   1:  PR[GP1:91,1] = PR[GP1:90,1] + -15.770;
   1:  PR[GP1:91,2] = PR[GP1:90,2] + -15.065;
   1:L PR[91] 10mm/sec CNT100;
   1:  PR[GP1:91,1] = PR[GP1:90,1] + -15.094;
   1:  PR[GP1:91,2] = PR[GP1:90,2] + -15.115;
   1:  PR[GP1:91,3] = PR[GP1:90,3] + 48.400;
   1:L PR[91] 10mm/sec CNT100;
   1:  PR[GP1:91,1] = PR[GP1:90,1] + -12.204;
   1:  PR[GP1:91,2] = PR[GP1:90,2] + -18.068;
   1:L PR[91] 10mm/sec CNT100;
   1:  PR[GP1:91,1] = PR[GP1:90,1] + -12.047;
   1:  PR[GP1:91,2] = PR[GP1:90,2] + -18.203;
   1:L PR[91] 10mm/sec CNT100;
   1:  PR[GP1:91,1] = PR[GP1:90,1] + -10.939;
   1:  PR[GP1:91,2] = PR[GP1:90,2] + -18.959;
   1:L PR[91] 10mm/sec CNT100;
   1:  PR[GP1:91,1] = PR[GP1:90,1] + -8.236;
   1:  PR[GP1:91,2] = PR[GP1:90,2] + -20.991;
   1:L PR[91] 10mm/sec CNT100;
   1:  PR[GP1:91,1] = PR[GP1:90,1] + -7.444;
   1:  PR[GP1:91,2] = PR[GP1:90,2] + -21.525;
   1:L PR[91] 10mm/sec CNT100;
   1:  PR[GP1:91,1] = PR[GP1:90,1] + -4.180;
   1:  PR[GP1:91,2] = PR[GP1:90,2] + -23.163;
   1:L PR[91] 10mm/sec CNT100;
   1:  PR[GP1:91,1] = PR[GP1:90,1] + -1.871;
   1:  PR[GP1:91,2] = PR[GP1:90,2] + -24.171;
   1:L PR[91] 10mm/sec CNT100;
   1:  PR[GP1:91,1] = PR[GP1:90,1] + 0.209;
   1:  PR[GP1:91,2] = PR[GP1:90,2] + -24.790;
   1:L PR[91] 10mm/sec CNT100;
   1:  PR[GP1:91,1] = PR[GP1:90,1] + 4.204;
   1:  PR[GP1:91,2] = PR[GP1:90,2] + -25.728;
   1:L PR[91] 10mm/sec CNT100;
   1:  PR[GP1:91,1] = PR[GP1:90,1] + 4.832;
   1:  PR[GP1:91,2] = PR[GP1:90,2] + -25.796;
   1:L PR[91] 10mm/sec CNT100;
   1:  PR[GP1:91,1] = PR[GP1:90,1] + 7.181;
   1:  PR[GP1:91,2] = PR[GP1:90,2] + -25.893;
   1:L PR[91] 10mm/sec CNT100;
   1:  PR[GP1:91,1] = PR[GP1:90,1] + 9.648;
   1:  PR[GP1:91,2] = PR[GP1:90,2] + -26.131;
   1:L PR[91] 10mm/sec CNT100;
   1:  PR[GP1:91,1] = PR[GP1:90,1] + 9.702;
   1:  PR[GP1:91,2] = PR[GP1:90,2] + -26.096;
   1:L PR[91] 10mm/sec CNT100;
   1:  PR[GP1:91,1] = PR[GP1:90,1] + 10.831;
   1:  PR[GP1:91,2] = PR[GP1:90,2] + -26.181;
   1:L PR[91] 10mm/sec CNT100;
   1:  PR[GP1:91,1] = PR[GP1:90,1] + 13.329;
   1:  PR[GP1:91,2] = PR[GP1:90,2] + -26.259;
   1:L PR[91] 10mm/sec CNT100;
   1:  PR[GP1:91,1] = PR[GP1:90,1] + 13.483;
   1:  PR[GP1:91,2] = PR[GP1:90,2] + -26.256;
   1:L PR[91] 10mm/sec CNT100;
   1:  PR[GP1:91,1] = PR[GP1:90,1] + 15.783;
   1:  PR[GP1:91,2] = PR[GP1:90,2] + -26.009;
   1:L PR[91] 10mm/sec CNT100;
   1:  PR[GP1:91,1] = PR[GP1:90,1] + 16.739;
   1:  PR[GP1:91,2] = PR[GP1:90,2] + -25.829;
   1:L PR[91] 10mm/sec CNT100;
   1:  PR[GP1:91,1] = PR[GP1:90,1] + 18.227;
   1:  PR[GP1:91,2] = PR[GP1:90,2] + -25.423;
   1:L PR[91] 10mm/sec CNT100;
   1:  PR[GP1:91,1] = PR[GP1:90,1] + 19.830;
   1:  PR[GP1:91,2] = PR[GP1:90,2] + -24.829;
   1:L PR[91] 10mm/sec CNT100;
   1:  PR[GP1:91,1] = PR[GP1:90,1] + 20.623;
   1:  PR[GP1:91,2] = PR[GP1:90,2] + -24.464;
   1:L PR[91] 10mm/sec CNT100;
   1:  PR[GP1:91,1] = PR[GP1:90,1] + 22.593;
   1:  PR[GP1:91,2] = PR[GP1:90,2] + -23.304;
   1:L PR[91] 10mm/sec CNT100;
   1:  PR[GP1:91,1] = PR[GP1:90,1] + 22.905;
   1:  PR[GP1:91,2] = PR[GP1:90,2] + -23.089;
   1:L PR[91] 10mm/sec CNT100;
   1:  PR[GP1:91,1] = PR[GP1:90,1] + 24.893;
   1:  PR[GP1:91,2] = PR[GP1:90,2] + -21.368;
   1:L PR[91] 10mm/sec CNT100;
   1:  PR[GP1:91,1] = PR[GP1:90,1] + 24.984;
   1:  PR[GP1:91,2] = PR[GP1:90,2] + -21.279;
   1:L PR[91] 10mm/sec CNT100;
   1:  PR[GP1:91,1] = PR[GP1:90,1] + 26.658;
   1:  PR[GP1:91,2] = PR[GP1:90,2] + -19.173;
   1:L PR[91] 10mm/sec CNT100;
   1:  PR[GP1:91,1] = PR[GP1:90,1] + 26.752;
   1:  PR[GP1:91,2] = PR[GP1:90,2] + -19.040;
   1:L PR[91] 10mm/sec CNT100;
   1:  PR[GP1:91,1] = PR[GP1:90,1] + 27.909;
   1:  PR[GP1:91,2] = PR[GP1:90,2] + -16.870;
   1:L PR[91] 10mm/sec CNT100;
   1:  PR[GP1:91,1] = PR[GP1:90,1] + 28.113;
   1:  PR[GP1:91,2] = PR[GP1:90,2] + -16.441;
   1:L PR[91] 10mm/sec CNT100;
   1:  PR[GP1:91,1] = PR[GP1:90,1] + 28.728;
   1:  PR[GP1:91,2] = PR[GP1:90,2] + -14.577;
   1:L PR[91] 10mm/sec CNT100;
   1:  PR[GP1:91,1] = PR[GP1:90,1] + 29.009;
   1:  PR[GP1:91,2] = PR[GP1:90,2] + -13.612;
   1:L PR[91] 10mm/sec CNT100;
   1:  PR[GP1:91,1] = PR[GP1:90,1] + 29.195;
   1:  PR[GP1:91,2] = PR[GP1:90,2] + -12.364;
   1:L PR[91] 10mm/sec CNT100;
   1:  PR[GP1:91,1] = PR[GP1:90,1] + 29.399;
   1:  PR[GP1:91,2] = PR[GP1:90,2] + -10.701;
   1:L PR[91] 10mm/sec CNT100;
   1:  PR[GP1:91,1] = PR[GP1:90,1] + 29.327;
   1:  PR[GP1:91,2] = PR[GP1:90,2] + -9.105;
   1:L PR[91] 10mm/sec CNT100;
   1:  PR[GP1:91,1] = PR[GP1:90,1] + 29.296;
   1:  PR[GP1:91,2] = PR[GP1:90,2] + -7.776;
   1:L PR[91] 10mm/sec CNT100;
   1:  PR[GP1:91,1] = PR[GP1:90,1] + 28.542;
   1:  PR[GP1:91,2] = PR[GP1:90,2] + -3.810;
   1:L PR[91] 10mm/sec CNT100;
   1:  PR[GP1:91,1] = PR[GP1:90,1] + 27.855;
   1:  PR[GP1:91,2] = PR[GP1:90,2] + -2.041;
   1:L PR[91] 10mm/sec CNT100;
   1:  PR[GP1:91,1] = PR[GP1:90,1] + 27.141;
   1:  PR[GP1:91,2] = PR[GP1:90,2] + -0.046;
   1:L PR[91] 10mm/sec CNT100;
   1:  PR[GP1:91,1] = PR[GP1:90,1] + 26.192;
   1:  PR[GP1:91,2] = PR[GP1:90,2] + 1.584;
   1:L PR[91] 10mm/sec CNT100;
   1:  PR[GP1:91,1] = PR[GP1:90,1] + 25.121;
   1:  PR[GP1:91,2] = PR[GP1:90,2] + 3.337;
   1:L PR[91] 10mm/sec CNT100;
   1:  PR[GP1:91,1] = PR[GP1:90,1] + 22.561;
   1:  PR[GP1:91,2] = PR[GP1:90,2] + 6.231;
   1:L PR[91] 10mm/sec CNT100;
   1:  PR[GP1:91,1] = PR[GP1:90,1] + 19.685;
   1:  PR[GP1:91,2] = PR[GP1:90,2] + 8.504;
   1:L PR[91] 10mm/sec CNT100;
   1:  PR[GP1:91,1] = PR[GP1:90,1] + 17.372;
   1:  PR[GP1:91,2] = PR[GP1:90,2] + 9.702;
   1:L PR[91] 10mm/sec CNT100;
   1:  PR[GP1:91,1] = PR[GP1:90,1] + 16.514;
   1:  PR[GP1:91,2] = PR[GP1:90,2] + 10.131;
   1:L PR[91] 10mm/sec CNT100;
   1:  PR[GP1:91,1] = PR[GP1:90,1] + 13.120;
   1:  PR[GP1:91,2] = PR[GP1:90,2] + 11.100;
   1:L PR[91] 10mm/sec CNT100;
   1:  PR[GP1:91,1] = PR[GP1:90,1] + 9.749;
   1:  PR[GP1:91,2] = PR[GP1:90,2] + 11.359;
   1:L PR[91] 10mm/sec CNT100;
   1:  PR[GP1:91,1] = PR[GP1:90,1] + 7.022;
   1:  PR[GP1:91,2] = PR[GP1:90,2] + 11.063;
   1:L PR[91] 10mm/sec CNT100;
   1:  PR[GP1:91,1] = PR[GP1:90,1] + 6.312;
   1:  PR[GP1:91,2] = PR[GP1:90,2] + 10.967;
   1:L PR[91] 10mm/sec CNT100;
   1:  PR[GP1:91,1] = PR[GP1:90,1] + 5.302;
   1:  PR[GP1:91,2] = PR[GP1:90,2] + 10.725;
   1:L PR[91] 10mm/sec CNT100;
   1:  PR[GP1:91,1] = PR[GP1:90,1] + 4.246;
   1:  PR[GP1:91,2] = PR[GP1:90,2] + 10.670;
   1:L PR[91] 10mm/sec CNT100;
   1:  PR[GP1:91,1] = PR[GP1:90,1] + 3.038;
   1:  PR[GP1:91,2] = PR[GP1:90,2] + 10.819;
   1:L PR[91] 10mm/sec CNT100;
   1:  PR[GP1:91,1] = PR[GP1:90,1] + 2.391;
   1:  PR[GP1:91,2] = PR[GP1:90,2] + 10.872;
   1:L PR[91] 10mm/sec CNT100;
   1:  PR[GP1:91,1] = PR[GP1:90,1] + 0.714;
   1:  PR[GP1:91,2] = PR[GP1:90,2] + 10.880;
   1:L PR[91] 10mm/sec CNT100;
   1:  PR[GP1:91,1] = PR[GP1:90,1] + -2.362;
   1:  PR[GP1:91,2] = PR[GP1:90,2] + 10.966;
   1:L PR[91] 10mm/sec CNT100;
   1:  PR[GP1:91,1] = PR[GP1:90,1] + -2.905;
   1:  PR[GP1:91,2] = PR[GP1:90,2] + 10.871;
   1:L PR[91] 10mm/sec CNT100;
   1:  PR[GP1:91,1] = PR[GP1:90,1] + -5.532;
   1:  PR[GP1:91,2] = PR[GP1:90,2] + 10.488;
   1:L PR[91] 10mm/sec CNT100;
   1:  PR[GP1:91,1] = PR[GP1:90,1] + -6.743;
   1:  PR[GP1:91,2] = PR[GP1:90,2] + 10.278;
   1:L PR[91] 10mm/sec CNT100;
   1:  PR[GP1:91,1] = PR[GP1:90,1] + -10.509;
   1:  PR[GP1:91,2] = PR[GP1:90,2] + 8.898;
   1:L PR[91] 10mm/sec CNT100;
   1:  PR[GP1:91,1] = PR[GP1:90,1] + -11.154;
   1:  PR[GP1:91,2] = PR[GP1:90,2] + 8.565;
   1:L PR[91] 10mm/sec CNT100;
   1:  PR[GP1:91,1] = PR[GP1:90,1] + -13.410;
   1:  PR[GP1:91,2] = PR[GP1:90,2] + 7.155;
   1:L PR[91] 10mm/sec CNT100;
   1:  PR[GP1:91,1] = PR[GP1:90,1] + -14.230;
   1:  PR[GP1:91,2] = PR[GP1:90,2] + 6.566;
   1:L PR[91] 10mm/sec CNT100;
   1:  PR[GP1:91,1] = PR[GP1:90,1] + -15.076;
   1:  PR[GP1:91,2] = PR[GP1:90,2] + 5.725;
   1:L PR[91] 10mm/sec CNT100;
   1:  PR[GP1:91,1] = PR[GP1:90,1] + -16.449;
   1:  PR[GP1:91,2] = PR[GP1:90,2] + 4.321;
   1:L PR[91] 10mm/sec CNT100;
   1:  PR[GP1:91,1] = PR[GP1:90,1] + -17.220;
   1:  PR[GP1:91,2] = PR[GP1:90,2] + 3.226;
   1:L PR[91] 10mm/sec CNT100;
   1:  PR[GP1:91,1] = PR[GP1:90,1] + -18.002;
   1:  PR[GP1:91,2] = PR[GP1:90,2] + 1.859;
   1:L PR[91] 10mm/sec CNT100;
   1:  PR[GP1:91,1] = PR[GP1:90,1] + -18.613;
   1:  PR[GP1:91,2] = PR[GP1:90,2] + 0.586;
   1:L PR[91] 10mm/sec CNT100;
   1:  PR[GP1:91,1] = PR[GP1:90,1] + -18.999;
   1:  PR[GP1:91,2] = PR[GP1:90,2] + -0.732;
   1:L PR[91] 10mm/sec CNT100;
   1:  PR[GP1:91,1] = PR[GP1:90,1] + -19.382;
   1:  PR[GP1:91,2] = PR[GP1:90,2] + -2.113;
   1:L PR[91] 10mm/sec CNT100;
   1:  PR[GP1:91,1] = PR[GP1:90,1] + -19.503;
   1:  PR[GP1:91,2] = PR[GP1:90,2] + -3.246;
   1:L PR[91] 10mm/sec CNT100;
   1:  PR[GP1:91,1] = PR[GP1:90,1] + -19.408;
   1:  PR[GP1:91,2] = PR[GP1:90,2] + -4.297;
   1:L PR[91] 10mm/sec CNT100;
   1:  PR[GP1:91,1] = PR[GP1:90,1] + -19.357;
   1:  PR[GP1:91,2] = PR[GP1:90,2] + -5.931;
   1:L PR[91] 10mm/sec CNT100;
   1:  PR[GP1:91,1] = PR[GP1:90,1] + -18.969;
   1:  PR[GP1:91,2] = PR[GP1:90,2] + -7.508;
   1:L PR[91] 10mm/sec CNT100;
   1:  PR[GP1:91,1] = PR[GP1:90,1] + -18.897;
   1:  PR[GP1:91,2] = PR[GP1:90,2] + -7.858;
   1:L PR[91] 10mm/sec CNT100;
   1:  PR[GP1:91,1] = PR[GP1:90,1] + -18.309;
   1:  PR[GP1:91,2] = PR[GP1:90,2] + -9.744;
   1:L PR[91] 10mm/sec CNT100;
   1:  PR[GP1:91,1] = PR[GP1:90,1] + -17.743;
   1:  PR[GP1:91,2] = PR[GP1:90,2] + -11.092;
   1:L PR[91] 10mm/sec CNT100;
   1:  PR[GP1:91,1] = PR[GP1:90,1] + -16.255;
   1:  PR[GP1:91,2] = PR[GP1:90,2] + -13.561;
   1:L PR[91] 10mm/sec CNT100;
   1:  PR[GP1:91,1] = PR[GP1:90,1] + -15.677;
   1:  PR[GP1:91,2] = PR[GP1:90,2] + -14.456;
   1:L PR[91] 10mm/sec CNT100;
   1:  PR[GP1:91,1] = PR[GP1:90,1] + -14.775;
   1:  PR[GP1:91,2] = PR[GP1:90,2] + -14.761;
   1:  PR[GP1:91,3] = PR[GP1:90,3] + 49.500;
   1:L PR[91] 10mm/sec CNT100;
   1:  PR[GP1:91,1] = PR[GP1:90,1] + -14.417;
   1:  PR[GP1:91,2] = PR[GP1:90,2] + -15.165;
   1:L PR[91] 10mm/sec CNT100;
   1:  PR[GP1:91,1] = PR[GP1:90,1] + -11.762;
   1:  PR[GP1:91,2] = PR[GP1:90,2] + -17.878;
   1:L PR[91] 10mm/sec CNT100;
   1:  PR[GP1:91,1] = PR[GP1:90,1] + -11.164;
   1:  PR[GP1:91,2] = PR[GP1:90,2] + -18.525;
   1:L PR[91] 10mm/sec CNT100;
   1:  PR[GP1:91,1] = PR[GP1:90,1] + -7.674;
   1:  PR[GP1:91,2] = PR[GP1:90,2] + -21.149;
   1:L PR[91] 10mm/sec CNT100;
   1:  PR[GP1:91,1] = PR[GP1:90,1] + -6.405;
   1:  PR[GP1:91,2] = PR[GP1:90,2] + -22.005;
   1:L PR[91] 10mm/sec CNT100;
   1:  PR[GP1:91,1] = PR[GP1:90,1] + -3.644;
   1:  PR[GP1:91,2] = PR[GP1:90,2] + -23.391;
   1:L PR[91] 10mm/sec CNT100;
   1:  PR[GP1:91,1] = PR[GP1:90,1] + -0.787;
   1:  PR[GP1:91,2] = PR[GP1:90,2] + -24.637;
   1:L PR[91] 10mm/sec CNT100;
   1:  PR[GP1:91,1] = PR[GP1:90,1] + 0.739;
   1:  PR[GP1:91,2] = PR[GP1:90,2] + -25.091;
   1:L PR[91] 10mm/sec CNT100;
   1:  PR[GP1:91,1] = PR[GP1:90,1] + 5.307;
   1:  PR[GP1:91,2] = PR[GP1:90,2] + -26.164;
   1:L PR[91] 10mm/sec CNT100;
   1:  PR[GP1:91,1] = PR[GP1:90,1] + 5.772;
   1:  PR[GP1:91,2] = PR[GP1:90,2] + -26.190;
   1:L PR[91] 10mm/sec CNT100;
   1:  PR[GP1:91,1] = PR[GP1:90,1] + 10.401;
   1:  PR[GP1:91,2] = PR[GP1:90,2] + -26.636;
   1:L PR[91] 10mm/sec CNT100;
   1:  PR[GP1:91,1] = PR[GP1:90,1] + 10.434;
   1:  PR[GP1:91,2] = PR[GP1:90,2] + -26.619;
   1:L PR[91] 10mm/sec CNT100;
   1:  PR[GP1:91,1] = PR[GP1:90,1] + 10.667;
   1:  PR[GP1:91,2] = PR[GP1:90,2] + -26.588;
   1:L PR[91] 10mm/sec CNT100;
   1:  PR[GP1:91,1] = PR[GP1:90,1] + 13.212;
   1:  PR[GP1:91,2] = PR[GP1:90,2] + -26.704;
   1:L PR[91] 10mm/sec CNT100;
   1:  PR[GP1:91,1] = PR[GP1:90,1] + 14.461;
   1:  PR[GP1:91,2] = PR[GP1:90,2] + -26.677;
   1:L PR[91] 10mm/sec CNT100;
   1:  PR[GP1:91,1] = PR[GP1:90,1] + 15.692;
   1:  PR[GP1:91,2] = PR[GP1:90,2] + -26.545;
   1:L PR[91] 10mm/sec CNT100;
   1:  PR[GP1:91,1] = PR[GP1:90,1] + 17.807;
   1:  PR[GP1:91,2] = PR[GP1:90,2] + -26.148;
   1:L PR[91] 10mm/sec CNT100;
   1:  PR[GP1:91,1] = PR[GP1:90,1] + 18.181;
   1:  PR[GP1:91,2] = PR[GP1:90,2] + -26.046;
   1:L PR[91] 10mm/sec CNT100;
   1:  PR[GP1:91,1] = PR[GP1:90,1] + 19.729;
   1:  PR[GP1:91,2] = PR[GP1:90,2] + -25.471;
   1:L PR[91] 10mm/sec CNT100;
   1:  PR[GP1:91,1] = PR[GP1:90,1] + 20.644;
   1:  PR[GP1:91,2] = PR[GP1:90,2] + -25.156;
   1:L PR[91] 10mm/sec CNT100;
   1:  PR[GP1:91,1] = PR[GP1:90,1] + 20.894;
   1:  PR[GP1:91,2] = PR[GP1:90,2] + -25.052;
   1:L PR[91] 10mm/sec CNT100;
   1:  PR[GP1:91,1] = PR[GP1:90,1] + 22.809;
   1:  PR[GP1:91,2] = PR[GP1:90,2] + -23.971;
   1:L PR[91] 10mm/sec CNT100;
   1:  PR[GP1:91,1] = PR[GP1:90,1] + 23.551;
   1:  PR[GP1:91,2] = PR[GP1:90,2] + -23.498;
   1:L PR[91] 10mm/sec CNT100;
   1:  PR[GP1:91,1] = PR[GP1:90,1] + 24.810;
   1:  PR[GP1:91,2] = PR[GP1:90,2] + -22.429;
   1:L PR[91] 10mm/sec CNT100;
   1:  PR[GP1:91,1] = PR[GP1:90,1] + 25.728;
   1:  PR[GP1:91,2] = PR[GP1:90,2] + -21.577;
   1:L PR[91] 10mm/sec CNT100;
   1:  PR[GP1:91,1] = PR[GP1:90,1] + 26.624;
   1:  PR[GP1:91,2] = PR[GP1:90,2] + -20.448;
   1:L PR[91] 10mm/sec CNT100;
   1:  PR[GP1:91,1] = PR[GP1:90,1] + 27.429;
   1:  PR[GP1:91,2] = PR[GP1:90,2] + -19.359;
   1:L PR[91] 10mm/sec CNT100;
   1:  PR[GP1:91,1] = PR[GP1:90,1] + 28.198;
   1:  PR[GP1:91,2] = PR[GP1:90,2] + -17.873;
   1:L PR[91] 10mm/sec CNT100;
   1:  PR[GP1:91,1] = PR[GP1:90,1] + 28.677;
   1:  PR[GP1:91,2] = PR[GP1:90,2] + -16.894;
   1:L PR[91] 10mm/sec CNT100;
   1:  PR[GP1:91,1] = PR[GP1:90,1] + 29.494;
   1:  PR[GP1:91,2] = PR[GP1:90,2] + -14.222;
   1:L PR[91] 10mm/sec CNT100;
   1:  PR[GP1:91,1] = PR[GP1:90,1] + 29.567;
   1:  PR[GP1:91,2] = PR[GP1:90,2] + -13.626;
   1:L PR[91] 10mm/sec CNT100;
   1:  PR[GP1:91,1] = PR[GP1:90,1] + 29.843;
   1:  PR[GP1:91,2] = PR[GP1:90,2] + -11.776;
   1:L PR[91] 10mm/sec CNT100;
   1:  PR[GP1:91,1] = PR[GP1:90,1] + 29.906;
   1:  PR[GP1:91,2] = PR[GP1:90,2] + -11.265;
   1:L PR[91] 10mm/sec CNT100;
   1:  PR[GP1:91,1] = PR[GP1:90,1] + 29.772;
   1:  PR[GP1:91,2] = PR[GP1:90,2] + -8.276;
   1:L PR[91] 10mm/sec CNT100;
   1:  PR[GP1:91,1] = PR[GP1:90,1] + 29.313;
   1:  PR[GP1:91,2] = PR[GP1:90,2] + -6.128;
   1:L PR[91] 10mm/sec CNT100;
   1:  PR[GP1:91,1] = PR[GP1:90,1] + 28.968;
   1:  PR[GP1:91,2] = PR[GP1:90,2] + -4.312;
   1:L PR[91] 10mm/sec CNT100;
   1:  PR[GP1:91,1] = PR[GP1:90,1] + 27.514;
   1:  PR[GP1:91,2] = PR[GP1:90,2] + -0.545;
   1:L PR[91] 10mm/sec CNT100;
   1:  PR[GP1:91,1] = PR[GP1:90,1] + 27.065;
   1:  PR[GP1:91,2] = PR[GP1:90,2] + 0.175;
   1:L PR[91] 10mm/sec CNT100;
   1:  PR[GP1:91,1] = PR[GP1:90,1] + 25.979;
   1:  PR[GP1:91,2] = PR[GP1:90,2] + 2.041;
   1:L PR[91] 10mm/sec CNT100;
   1:  PR[GP1:91,1] = PR[GP1:90,1] + 25.461;
   1:  PR[GP1:91,2] = PR[GP1:90,2] + 2.889;
   1:L PR[91] 10mm/sec CNT100;
   1:  PR[GP1:91,1] = PR[GP1:90,1] + 24.290;
   1:  PR[GP1:91,2] = PR[GP1:90,2] + 4.246;
   1:L PR[91] 10mm/sec CNT100;
   1:  PR[GP1:91,1] = PR[GP1:90,1] + 22.888;
   1:  PR[GP1:91,2] = PR[GP1:90,2] + 5.816;
   1:L PR[91] 10mm/sec CNT100;
   1:  PR[GP1:91,1] = PR[GP1:90,1] + 22.224;
   1:  PR[GP1:91,2] = PR[GP1:90,2] + 6.350;
   1:L PR[91] 10mm/sec CNT100;
   1:  PR[GP1:91,1] = PR[GP1:90,1] + 19.917;
   1:  PR[GP1:91,2] = PR[GP1:90,2] + 8.142;
   1:L PR[91] 10mm/sec CNT100;
   1:  PR[GP1:91,1] = PR[GP1:90,1] + 16.680;
   1:  PR[GP1:91,2] = PR[GP1:90,2] + 9.812;
   1:L PR[91] 10mm/sec CNT100;
   1:  PR[GP1:91,1] = PR[GP1:90,1] + 13.327;
   1:  PR[GP1:91,2] = PR[GP1:90,2] + 10.785;
   1:L PR[91] 10mm/sec CNT100;
   1:  PR[GP1:91,1] = PR[GP1:90,1] + 12.263;
   1:  PR[GP1:91,2] = PR[GP1:90,2] + 10.889;
   1:L PR[91] 10mm/sec CNT100;
   1:  PR[GP1:91,1] = PR[GP1:90,1] + 9.919;
   1:  PR[GP1:91,2] = PR[GP1:90,2] + 11.069;
   1:L PR[91] 10mm/sec CNT100;
   1:  PR[GP1:91,1] = PR[GP1:90,1] + 6.422;
   1:  PR[GP1:91,2] = PR[GP1:90,2] + 10.685;
   1:L PR[91] 10mm/sec CNT100;
   1:  PR[GP1:91,1] = PR[GP1:90,1] + 5.657;
   1:  PR[GP1:91,2] = PR[GP1:90,2] + 10.509;
   1:L PR[91] 10mm/sec CNT100;
   1:  PR[GP1:91,1] = PR[GP1:90,1] + 4.669;
   1:  PR[GP1:91,2] = PR[GP1:90,2] + 10.459;
   1:L PR[91] 10mm/sec CNT100;
   1:  PR[GP1:91,1] = PR[GP1:90,1] + 3.629;
   1:  PR[GP1:91,2] = PR[GP1:90,2] + 10.568;
   1:L PR[91] 10mm/sec CNT100;
   1:  PR[GP1:91,1] = PR[GP1:90,1] + 3.132;
   1:  PR[GP1:91,2] = PR[GP1:90,2] + 10.596;
   1:L PR[91] 10mm/sec CNT100;
   1:  PR[GP1:91,1] = PR[GP1:90,1] + 1.112;
   1:  PR[GP1:91,2] = PR[GP1:90,2] + 10.600;
   1:L PR[91] 10mm/sec CNT100;
   1:  PR[GP1:91,1] = PR[GP1:90,1] + -1.522;
   1:  PR[GP1:91,2] = PR[GP1:90,2] + 10.674;
   1:L PR[91] 10mm/sec CNT100;
   1:  PR[GP1:91,1] = PR[GP1:90,1] + -2.503;
   1:  PR[GP1:91,2] = PR[GP1:90,2] + 10.503;
   1:L PR[91] 10mm/sec CNT100;
   1:  PR[GP1:91,1] = PR[GP1:90,1] + -5.863;
   1:  PR[GP1:91,2] = PR[GP1:90,2] + 10.013;
   1:L PR[91] 10mm/sec CNT100;
   1:  PR[GP1:91,1] = PR[GP1:90,1] + -7.016;
   1:  PR[GP1:91,2] = PR[GP1:90,2] + 9.606;
   1:L PR[91] 10mm/sec CNT100;
   1:  PR[GP1:91,1] = PR[GP1:90,1] + -9.727;
   1:  PR[GP1:91,2] = PR[GP1:90,2] + 8.610;
   1:L PR[91] 10mm/sec CNT100;
   1:  PR[GP1:91,1] = PR[GP1:90,1] + -10.037;
   1:  PR[GP1:91,2] = PR[GP1:90,2] + 8.449;
   1:L PR[91] 10mm/sec CNT100;
   1:  PR[GP1:91,1] = PR[GP1:90,1] + -12.742;
   1:  PR[GP1:91,2] = PR[GP1:90,2] + 6.760;
   1:L PR[91] 10mm/sec CNT100;
   1:  PR[GP1:91,1] = PR[GP1:90,1] + -13.296;
   1:  PR[GP1:91,2] = PR[GP1:90,2] + 6.362;
   1:L PR[91] 10mm/sec CNT100;
   1:  PR[GP1:91,1] = PR[GP1:90,1] + -15.633;
   1:  PR[GP1:91,2] = PR[GP1:90,2] + 3.989;
   1:L PR[91] 10mm/sec CNT100;
   1:  PR[GP1:91,1] = PR[GP1:90,1] + -16.206;
   1:  PR[GP1:91,2] = PR[GP1:90,2] + 3.175;
   1:L PR[91] 10mm/sec CNT100;
   1:  PR[GP1:91,1] = PR[GP1:90,1] + -17.234;
   1:  PR[GP1:91,2] = PR[GP1:90,2] + 1.377;
   1:L PR[91] 10mm/sec CNT100;
   1:  PR[GP1:91,1] = PR[GP1:90,1] + -17.703;
   1:  PR[GP1:91,2] = PR[GP1:90,2] + 0.402;
   1:L PR[91] 10mm/sec CNT100;
   1:  PR[GP1:91,1] = PR[GP1:90,1] + -17.999;
   1:  PR[GP1:91,2] = PR[GP1:90,2] + -0.611;
   1:L PR[91] 10mm/sec CNT100;
   1:  PR[GP1:91,1] = PR[GP1:90,1] + -18.515;
   1:  PR[GP1:91,2] = PR[GP1:90,2] + -2.471;
   1:L PR[91] 10mm/sec CNT100;
   1:  PR[GP1:91,1] = PR[GP1:90,1] + -18.605;
   1:  PR[GP1:91,2] = PR[GP1:90,2] + -3.323;
   1:L PR[91] 10mm/sec CNT100;
   1:  PR[GP1:91,1] = PR[GP1:90,1] + -18.533;
   1:  PR[GP1:91,2] = PR[GP1:90,2] + -4.127;
   1:L PR[91] 10mm/sec CNT100;
   1:  PR[GP1:91,1] = PR[GP1:90,1] + -18.467;
   1:  PR[GP1:91,2] = PR[GP1:90,2] + -6.252;
   1:L PR[91] 10mm/sec CNT100;
   1:  PR[GP1:91,1] = PR[GP1:90,1] + -18.182;
   1:  PR[GP1:91,2] = PR[GP1:90,2] + -7.409;
   1:L PR[91] 10mm/sec CNT100;
   1:  PR[GP1:91,1] = PR[GP1:90,1] + -18.092;
   1:  PR[GP1:91,2] = PR[GP1:90,2] + -7.848;
   1:L PR[91] 10mm/sec CNT100;
   1:  PR[GP1:91,1] = PR[GP1:90,1] + -17.358;
   1:  PR[GP1:91,2] = PR[GP1:90,2] + -10.202;
   1:L PR[91] 10mm/sec CNT100;
   1:  PR[GP1:91,1] = PR[GP1:90,1] + -16.925;
   1:  PR[GP1:91,2] = PR[GP1:90,2] + -11.233;
   1:L PR[91] 10mm/sec CNT100;
   1:  PR[GP1:91,1] = PR[GP1:90,1] + -15.134;
   1:  PR[GP1:91,2] = PR[GP1:90,2] + -14.204;
   1:L PR[91] 10mm/sec CNT100;
   1:  PR[GP1:91,1] = PR[GP1:90,1] + -13.873;
   1:  PR[GP1:91,2] = PR[GP1:90,2] + -15.065;
   1:  PR[GP1:91,3] = PR[GP1:90,3] + 50.600;
   1:L PR[91] 10mm/sec CNT100;
   1:  PR[GP1:91,1] = PR[GP1:90,1] + -13.740;
   1:  PR[GP1:91,2] = PR[GP1:90,2] + -15.215;
   1:L PR[91] 10mm/sec CNT100;
   1:  PR[GP1:91,1] = PR[GP1:90,1] + -12.572;
   1:  PR[GP1:91,2] = PR[GP1:90,2] + -16.408;
   1:L PR[91] 10mm/sec CNT100;
   1:  PR[GP1:91,1] = PR[GP1:90,1] + -10.658;
   1:  PR[GP1:91,2] = PR[GP1:90,2] + -18.523;
   1:L PR[91] 10mm/sec CNT100;
   1:  PR[GP1:91,1] = PR[GP1:90,1] + -10.181;
   1:  PR[GP1:91,2] = PR[GP1:90,2] + -19.000;
   1:L PR[91] 10mm/sec CNT100;
   1:  PR[GP1:91,1] = PR[GP1:90,1] + -7.112;
   1:  PR[GP1:91,2] = PR[GP1:90,2] + -21.308;
   1:L PR[91] 10mm/sec CNT100;
   1:  PR[GP1:91,1] = PR[GP1:90,1] + -5.365;
   1:  PR[GP1:91,2] = PR[GP1:90,2] + -22.485;
   1:L PR[91] 10mm/sec CNT100;
   1:  PR[GP1:91,1] = PR[GP1:90,1] + -3.108;
   1:  PR[GP1:91,2] = PR[GP1:90,2] + -23.618;
   1:L PR[91] 10mm/sec CNT100;
   1:  PR[GP1:91,1] = PR[GP1:90,1] + 0.296;
   1:  PR[GP1:91,2] = PR[GP1:90,2] + -25.103;
   1:L PR[91] 10mm/sec CNT100;
   1:  PR[GP1:91,1] = PR[GP1:90,1] + 1.269;
   1:  PR[GP1:91,2] = PR[GP1:90,2] + -25.392;
   1:L PR[91] 10mm/sec CNT100;
   1:  PR[GP1:91,1] = PR[GP1:90,1] + 4.599;
   1:  PR[GP1:91,2] = PR[GP1:90,2] + -26.175;
   1:L PR[91] 10mm/sec CNT100;
   1:  PR[GP1:91,1] = PR[GP1:90,1] + 6.163;
   1:  PR[GP1:91,2] = PR[GP1:90,2] + -26.632;
   1:L PR[91] 10mm/sec CNT100;
   1:  PR[GP1:91,1] = PR[GP1:90,1] + 6.679;
   1:  PR[GP1:91,2] = PR[GP1:90,2] + -26.710;
   1:L PR[91] 10mm/sec CNT100;
   1:  PR[GP1:91,1] = PR[GP1:90,1] + 11.123;
   1:  PR[GP1:91,2] = PR[GP1:90,2] + -27.139;
   1:L PR[91] 10mm/sec CNT100;
   1:  PR[GP1:91,1] = PR[GP1:90,1] + 11.142;
   1:  PR[GP1:91,2] = PR[GP1:90,2] + -27.128;
   1:L PR[91] 10mm/sec CNT100;
   1:  PR[GP1:91,1] = PR[GP1:90,1] + 11.547;
   1:  PR[GP1:91,2] = PR[GP1:90,2] + -27.075;
   1:L PR[91] 10mm/sec CNT100;
   1:  PR[GP1:91,1] = PR[GP1:90,1] + 13.092;
   1:  PR[GP1:91,2] = PR[GP1:90,2] + -27.149;
   1:L PR[91] 10mm/sec CNT100;
   1:  PR[GP1:91,1] = PR[GP1:90,1] + 15.439;
   1:  PR[GP1:91,2] = PR[GP1:90,2] + -27.099;
   1:L PR[91] 10mm/sec CNT100;
   1:  PR[GP1:91,1] = PR[GP1:90,1] + 15.600;
   1:  PR[GP1:91,2] = PR[GP1:90,2] + -27.081;
   1:L PR[91] 10mm/sec CNT100;
   1:  PR[GP1:91,1] = PR[GP1:90,1] + 16.227;
   1:  PR[GP1:91,2] = PR[GP1:90,2] + -26.964;
   1:L PR[91] 10mm/sec CNT100;
   1:  PR[GP1:91,1] = PR[GP1:90,1] + 18.101;
   1:  PR[GP1:91,2] = PR[GP1:90,2] + -26.662;
   1:L PR[91] 10mm/sec CNT100;
   1:  PR[GP1:91,1] = PR[GP1:90,1] + 18.852;
   1:  PR[GP1:91,2] = PR[GP1:90,2] + -26.488;
   1:L PR[91] 10mm/sec CNT100;
   1:  PR[GP1:91,1] = PR[GP1:90,1] + 20.377;
   1:  PR[GP1:91,2] = PR[GP1:90,2] + -25.963;
   1:L PR[91] 10mm/sec CNT100;
   1:  PR[GP1:91,1] = PR[GP1:90,1] + 21.895;
   1:  PR[GP1:91,2] = PR[GP1:90,2] + -25.334;
   1:L PR[91] 10mm/sec CNT100;
   1:  PR[GP1:91,1] = PR[GP1:90,1] + 22.513;
   1:  PR[GP1:91,2] = PR[GP1:90,2] + -24.985;
   1:L PR[91] 10mm/sec CNT100;
   1:  PR[GP1:91,1] = PR[GP1:90,1] + 24.455;
   1:  PR[GP1:91,2] = PR[GP1:90,2] + -23.748;
   1:L PR[91] 10mm/sec CNT100;
   1:  PR[GP1:91,1] = PR[GP1:90,1] + 26.511;
   1:  PR[GP1:91,2] = PR[GP1:90,2] + -21.868;
   1:L PR[91] 10mm/sec CNT100;
   1:  PR[GP1:91,1] = PR[GP1:90,1] + 28.157;
   1:  PR[GP1:91,2] = PR[GP1:90,2] + -19.646;
   1:L PR[91] 10mm/sec CNT100;
   1:  PR[GP1:91,1] = PR[GP1:90,1] + 29.365;
   1:  PR[GP1:91,2] = PR[GP1:90,2] + -17.147;
   1:L PR[91] 10mm/sec CNT100;
   1:  PR[GP1:91,1] = PR[GP1:90,1] + 30.137;
   1:  PR[GP1:91,2] = PR[GP1:90,2] + -14.511;
   1:L PR[91] 10mm/sec CNT100;
   1:  PR[GP1:91,1] = PR[GP1:90,1] + 30.465;
   1:  PR[GP1:91,2] = PR[GP1:90,2] + -11.719;
   1:L PR[91] 10mm/sec CNT100;
   1:  PR[GP1:91,1] = PR[GP1:90,1] + 30.345;
   1:  PR[GP1:91,2] = PR[GP1:90,2] + -9.944;
   1:L PR[91] 10mm/sec CNT100;
   1:  PR[GP1:91,1] = PR[GP1:90,1] + 30.285;
   1:  PR[GP1:91,2] = PR[GP1:90,2] + -8.738;
   1:L PR[91] 10mm/sec CNT100;
   1:  PR[GP1:91,1] = PR[GP1:90,1] + 29.440;
   1:  PR[GP1:91,2] = PR[GP1:90,2] + -4.805;
   1:L PR[91] 10mm/sec CNT100;
   1:  PR[GP1:91,1] = PR[GP1:90,1] + 28.977;
   1:  PR[GP1:91,2] = PR[GP1:90,2] + -3.685;
   1:L PR[91] 10mm/sec CNT100;
   1:  PR[GP1:91,1] = PR[GP1:90,1] + 27.958;
   1:  PR[GP1:91,2] = PR[GP1:90,2] + -1.020;
   1:L PR[91] 10mm/sec CNT100;
   1:  PR[GP1:91,1] = PR[GP1:90,1] + 27.249;
   1:  PR[GP1:91,2] = PR[GP1:90,2] + 0.144;
   1:L PR[91] 10mm/sec CNT100;
   1:  PR[GP1:91,1] = PR[GP1:90,1] + 25.807;
   1:  PR[GP1:91,2] = PR[GP1:90,2] + 2.434;
   1:L PR[91] 10mm/sec CNT100;
   1:  PR[GP1:91,1] = PR[GP1:90,1] + 23.950;
   1:  PR[GP1:91,2] = PR[GP1:90,2] + 4.585;
   1:L PR[91] 10mm/sec CNT100;
   1:  PR[GP1:91,1] = PR[GP1:90,1] + 23.225;
   1:  PR[GP1:91,2] = PR[GP1:90,2] + 5.397;
   1:L PR[91] 10mm/sec CNT100;
   1:  PR[GP1:91,1] = PR[GP1:90,1] + 21.792;
   1:  PR[GP1:91,2] = PR[GP1:90,2] + 6.548;
   1:L PR[91] 10mm/sec CNT100;
   1:  PR[GP1:91,1] = PR[GP1:90,1] + 20.237;
   1:  PR[GP1:91,2] = PR[GP1:90,2] + 7.756;
   1:L PR[91] 10mm/sec CNT100;
   1:  PR[GP1:91,1] = PR[GP1:90,1] + 19.198;
   1:  PR[GP1:91,2] = PR[GP1:90,2] + 8.311;
   1:L PR[91] 10mm/sec CNT100;
   1:  PR[GP1:91,1] = PR[GP1:90,1] + 16.975;
   1:  PR[GP1:91,2] = PR[GP1:90,2] + 9.455;
   1:L PR[91] 10mm/sec CNT100;
   1:  PR[GP1:91,1] = PR[GP1:90,1] + 15.892;
   1:  PR[GP1:91,2] = PR[GP1:90,2] + 9.786;
   1:L PR[91] 10mm/sec CNT100;
   1:  PR[GP1:91,1] = PR[GP1:90,1] + 13.573;
   1:  PR[GP1:91,2] = PR[GP1:90,2] + 10.459;
   1:L PR[91] 10mm/sec CNT100;
   1:  PR[GP1:91,1] = PR[GP1:90,1] + 11.016;
   1:  PR[GP1:91,2] = PR[GP1:90,2] + 10.708;
   1:L PR[91] 10mm/sec CNT100;
   1:  PR[GP1:91,1] = PR[GP1:90,1] + 10.090;
   1:  PR[GP1:91,2] = PR[GP1:90,2] + 10.779;
   1:L PR[91] 10mm/sec CNT100;
   1:  PR[GP1:91,1] = PR[GP1:90,1] + 6.558;
   1:  PR[GP1:91,2] = PR[GP1:90,2] + 10.384;
   1:L PR[91] 10mm/sec CNT100;
   1:  PR[GP1:91,1] = PR[GP1:90,1] + 6.024;
   1:  PR[GP1:91,2] = PR[GP1:90,2] + 10.279;
   1:L PR[91] 10mm/sec CNT100;
   1:  PR[GP1:91,1] = PR[GP1:90,1] + 5.107;
   1:  PR[GP1:91,2] = PR[GP1:90,2] + 10.233;
   1:L PR[91] 10mm/sec CNT100;
   1:  PR[GP1:91,1] = PR[GP1:90,1] + 4.603;
   1:  PR[GP1:91,2] = PR[GP1:90,2] + 10.281;
   1:L PR[91] 10mm/sec CNT100;
   1:  PR[GP1:91,1] = PR[GP1:90,1] + 3.983;
   1:  PR[GP1:91,2] = PR[GP1:90,2] + 10.316;
   1:L PR[91] 10mm/sec CNT100;
   1:  PR[GP1:91,1] = PR[GP1:90,1] + 1.509;
   1:  PR[GP1:91,2] = PR[GP1:90,2] + 10.321;
   1:L PR[91] 10mm/sec CNT100;
   1:  PR[GP1:91,1] = PR[GP1:90,1] + -0.682;
   1:  PR[GP1:91,2] = PR[GP1:90,2] + 10.383;
   1:L PR[91] 10mm/sec CNT100;
   1:  PR[GP1:91,1] = PR[GP1:90,1] + -2.101;
   1:  PR[GP1:91,2] = PR[GP1:90,2] + 10.135;
   1:L PR[91] 10mm/sec CNT100;
   1:  PR[GP1:91,1] = PR[GP1:90,1] + -5.022;
   1:  PR[GP1:91,2] = PR[GP1:90,2] + 9.709;
   1:L PR[91] 10mm/sec CNT100;
   1:  PR[GP1:91,1] = PR[GP1:90,1] + -5.567;
   1:  PR[GP1:91,2] = PR[GP1:90,2] + 9.500;
   1:L PR[91] 10mm/sec CNT100;
   1:  PR[GP1:91,1] = PR[GP1:90,1] + -8.924;
   1:  PR[GP1:91,2] = PR[GP1:90,2] + 8.328;
   1:L PR[91] 10mm/sec CNT100;
   1:  PR[GP1:91,1] = PR[GP1:90,1] + -12.074;
   1:  PR[GP1:91,2] = PR[GP1:90,2] + 6.365;
   1:L PR[91] 10mm/sec CNT100;
   1:  PR[GP1:91,1] = PR[GP1:90,1] + -12.364;
   1:  PR[GP1:91,2] = PR[GP1:90,2] + 6.156;
   1:L PR[91] 10mm/sec CNT100;
   1:  PR[GP1:91,1] = PR[GP1:90,1] + -14.816;
   1:  PR[GP1:91,2] = PR[GP1:90,2] + 3.658;
   1:L PR[91] 10mm/sec CNT100;
   1:  PR[GP1:91,1] = PR[GP1:90,1] + -15.192;
   1:  PR[GP1:91,2] = PR[GP1:90,2] + 3.124;
   1:L PR[91] 10mm/sec CNT100;
   1:  PR[GP1:91,1] = PR[GP1:90,1] + -16.466;
   1:  PR[GP1:91,2] = PR[GP1:90,2] + 0.896;
   1:L PR[91] 10mm/sec CNT100;
   1:  PR[GP1:91,1] = PR[GP1:90,1] + -16.790;
   1:  PR[GP1:91,2] = PR[GP1:90,2] + 0.221;
   1:L PR[91] 10mm/sec CNT100;
   1:  PR[GP1:91,1] = PR[GP1:90,1] + -17.647;
   1:  PR[GP1:91,2] = PR[GP1:90,2] + -2.831;
   1:L PR[91] 10mm/sec CNT100;
   1:  PR[GP1:91,1] = PR[GP1:90,1] + -17.708;
   1:  PR[GP1:91,2] = PR[GP1:90,2] + -3.399;
   1:L PR[91] 10mm/sec CNT100;
   1:  PR[GP1:91,1] = PR[GP1:90,1] + -17.658;
   1:  PR[GP1:91,2] = PR[GP1:90,2] + -3.957;
   1:L PR[91] 10mm/sec CNT100;
   1:  PR[GP1:91,1] = PR[GP1:90,1] + -17.576;
   1:  PR[GP1:91,2] = PR[GP1:90,2] + -6.574;
   1:L PR[91] 10mm/sec CNT100;
   1:  PR[GP1:91,1] = PR[GP1:90,1] + -17.395;
   1:  PR[GP1:91,2] = PR[GP1:90,2] + -7.310;
   1:L PR[91] 10mm/sec CNT100;
   1:  PR[GP1:91,1] = PR[GP1:90,1] + -17.287;
   1:  PR[GP1:91,2] = PR[GP1:90,2] + -7.838;
   1:L PR[91] 10mm/sec CNT100;
   1:  PR[GP1:91,1] = PR[GP1:90,1] + -16.407;
   1:  PR[GP1:91,2] = PR[GP1:90,2] + -10.661;
   1:L PR[91] 10mm/sec CNT100;
   1:  PR[GP1:91,1] = PR[GP1:90,1] + -16.107;
   1:  PR[GP1:91,2] = PR[GP1:90,2] + -11.374;
   1:L PR[91] 10mm/sec CNT100;
   1:  PR[GP1:91,1] = PR[GP1:90,1] + -14.012;
   1:  PR[GP1:91,2] = PR[GP1:90,2] + -14.849;
   1:L PR[91] 10mm/sec CNT100;
   1:  PR[GP1:91,1] = PR[GP1:90,1] + -12.952;
   1:  PR[GP1:91,2] = PR[GP1:90,2] + -15.415;
   1:  PR[GP1:91,3] = PR[GP1:90,3] + 51.700;
   1:L PR[91] 10mm/sec CNT100;
   1:  PR[GP1:91,1] = PR[GP1:90,1] + -10.051;
   1:  PR[GP1:91,2] = PR[GP1:90,2] + -18.620;
   1:L PR[91] 10mm/sec CNT100;
   1:  PR[GP1:91,1] = PR[GP1:90,1] + -9.188;
   1:  PR[GP1:91,2] = PR[GP1:90,2] + -19.482;
   1:L PR[91] 10mm/sec CNT100;
   1:  PR[GP1:91,1] = PR[GP1:90,1] + -6.550;
   1:  PR[GP1:91,2] = PR[GP1:90,2] + -21.466;
   1:L PR[91] 10mm/sec CNT100;
   1:  PR[GP1:91,1] = PR[GP1:90,1] + -4.326;
   1:  PR[GP1:91,2] = PR[GP1:90,2] + -22.965;
   1:L PR[91] 10mm/sec CNT100;
   1:  PR[GP1:91,1] = PR[GP1:90,1] + -2.572;
   1:  PR[GP1:91,2] = PR[GP1:90,2] + -23.846;
   1:L PR[91] 10mm/sec CNT100;
   1:  PR[GP1:91,1] = PR[GP1:90,1] + 1.379;
   1:  PR[GP1:91,2] = PR[GP1:90,2] + -25.569;
   1:L PR[91] 10mm/sec CNT100;
   1:  PR[GP1:91,1] = PR[GP1:90,1] + 1.799;
   1:  PR[GP1:91,2] = PR[GP1:90,2] + -25.694;
   1:L PR[91] 10mm/sec CNT100;
   1:  PR[GP1:91,1] = PR[GP1:90,1] + 3.339;
   1:  PR[GP1:91,2] = PR[GP1:90,2] + -26.056;
   1:L PR[91] 10mm/sec CNT100;
   1:  PR[GP1:91,1] = PR[GP1:90,1] + 6.893;
   1:  PR[GP1:91,2] = PR[GP1:90,2] + -27.096;
   1:L PR[91] 10mm/sec CNT100;
   1:  PR[GP1:91,1] = PR[GP1:90,1] + 8.132;
   1:  PR[GP1:91,2] = PR[GP1:90,2] + -27.283;
   1:L PR[91] 10mm/sec CNT100;
   1:  PR[GP1:91,1] = PR[GP1:90,1] + 11.845;
   1:  PR[GP1:91,2] = PR[GP1:90,2] + -27.641;
   1:L PR[91] 10mm/sec CNT100;
   1:  PR[GP1:91,1] = PR[GP1:90,1] + 11.850;
   1:  PR[GP1:91,2] = PR[GP1:90,2] + -27.638;
   1:L PR[91] 10mm/sec CNT100;
   1:  PR[GP1:91,1] = PR[GP1:90,1] + 12.214;
   1:  PR[GP1:91,2] = PR[GP1:90,2] + -27.591;
   1:L PR[91] 10mm/sec CNT100;
   1:  PR[GP1:91,1] = PR[GP1:90,1] + 12.567;
   1:  PR[GP1:91,2] = PR[GP1:90,2] + -27.578;
   1:L PR[91] 10mm/sec CNT100;
   1:  PR[GP1:91,1] = PR[GP1:90,1] + 12.974;
   1:  PR[GP1:91,2] = PR[GP1:90,2] + -27.594;
   1:L PR[91] 10mm/sec CNT100;
   1:  PR[GP1:91,1] = PR[GP1:90,1] + 15.512;
   1:  PR[GP1:91,2] = PR[GP1:90,2] + -27.590;
   1:L PR[91] 10mm/sec CNT100;
   1:  PR[GP1:91,1] = PR[GP1:90,1] + 16.534;
   1:  PR[GP1:91,2] = PR[GP1:90,2] + -27.521;
   1:L PR[91] 10mm/sec CNT100;
   1:  PR[GP1:91,1] = PR[GP1:90,1] + 17.878;
   1:  PR[GP1:91,2] = PR[GP1:90,2] + -27.304;
   1:L PR[91] 10mm/sec CNT100;
   1:  PR[GP1:91,1] = PR[GP1:90,1] + 19.926;
   1:  PR[GP1:91,2] = PR[GP1:90,2] + -26.831;
   1:L PR[91] 10mm/sec CNT100;
   1:  PR[GP1:91,1] = PR[GP1:90,1] + 22.614;
   1:  PR[GP1:91,2] = PR[GP1:90,2] + -25.782;
   1:L PR[91] 10mm/sec CNT100;
   1:  PR[GP1:91,1] = PR[GP1:90,1] + 23.567;
   1:  PR[GP1:91,2] = PR[GP1:90,2] + -25.223;
   1:L PR[91] 10mm/sec CNT100;
   1:  PR[GP1:91,1] = PR[GP1:90,1] + 24.980;
   1:  PR[GP1:91,2] = PR[GP1:90,2] + -24.355;
   1:L PR[91] 10mm/sec CNT100;
   1:  PR[GP1:91,1] = PR[GP1:90,1] + 26.472;
   1:  PR[GP1:91,2] = PR[GP1:90,2] + -23.047;
   1:L PR[91] 10mm/sec CNT100;
   1:  PR[GP1:91,1] = PR[GP1:90,1] + 27.065;
   1:  PR[GP1:91,2] = PR[GP1:90,2] + -22.506;
   1:L PR[91] 10mm/sec CNT100;
   1:  PR[GP1:91,1] = PR[GP1:90,1] + 28.774;
   1:  PR[GP1:91,2] = PR[GP1:90,2] + -20.254;
   1:L PR[91] 10mm/sec CNT100;
   1:  PR[GP1:91,1] = PR[GP1:90,1] + 30.029;
   1:  PR[GP1:91,2] = PR[GP1:90,2] + -17.681;
   1:L PR[91] 10mm/sec CNT100;
   1:  PR[GP1:91,1] = PR[GP1:90,1] + 30.800;
   1:  PR[GP1:91,2] = PR[GP1:90,2] + -14.904;
   1:L PR[91] 10mm/sec CNT100;
   1:  PR[GP1:91,1] = PR[GP1:90,1] + 31.005;
   1:  PR[GP1:91,2] = PR[GP1:90,2] + -12.700;
   1:L PR[91] 10mm/sec CNT100;
   1:  PR[GP1:91,1] = PR[GP1:90,1] + 31.078;
   1:  PR[GP1:91,2] = PR[GP1:90,2] + -12.051;
   1:L PR[91] 10mm/sec CNT100;
   1:  PR[GP1:91,1] = PR[GP1:90,1] + 30.859;
   1:  PR[GP1:91,2] = PR[GP1:90,2] + -9.159;
   1:L PR[91] 10mm/sec CNT100;
   1:  PR[GP1:91,1] = PR[GP1:90,1] + 30.309;
   1:  PR[GP1:91,2] = PR[GP1:90,2] + -6.874;
   1:L PR[91] 10mm/sec CNT100;
   1:  PR[GP1:91,1] = PR[GP1:90,1] + 29.956;
   1:  PR[GP1:91,2] = PR[GP1:90,2] + -5.252;
   1:L PR[91] 10mm/sec CNT100;
   1:  PR[GP1:91,1] = PR[GP1:90,1] + 28.410;
   1:  PR[GP1:91,2] = PR[GP1:90,2] + -1.506;
   1:L PR[91] 10mm/sec CNT100;
   1:  PR[GP1:91,1] = PR[GP1:90,1] + 27.112;
   1:  PR[GP1:91,2] = PR[GP1:90,2] + 0.624;
   1:L PR[91] 10mm/sec CNT100;
   1:  PR[GP1:91,1] = PR[GP1:90,1] + 26.262;
   1:  PR[GP1:91,2] = PR[GP1:90,2] + 1.974;
   1:L PR[91] 10mm/sec CNT100;
   1:  PR[GP1:91,1] = PR[GP1:90,1] + 23.563;
   1:  PR[GP1:91,2] = PR[GP1:90,2] + 4.977;
   1:L PR[91] 10mm/sec CNT100;
   1:  PR[GP1:91,1] = PR[GP1:90,1] + 21.360;
   1:  PR[GP1:91,2] = PR[GP1:90,2] + 6.747;
   1:L PR[91] 10mm/sec CNT100;
   1:  PR[GP1:91,1] = PR[GP1:90,1] + 20.562;
   1:  PR[GP1:91,2] = PR[GP1:90,2] + 7.367;
   1:L PR[91] 10mm/sec CNT100;
   1:  PR[GP1:91,1] = PR[GP1:90,1] + 18.653;
   1:  PR[GP1:91,2] = PR[GP1:90,2] + 8.385;
   1:L PR[91] 10mm/sec CNT100;
   1:  PR[GP1:91,1] = PR[GP1:90,1] + 17.274;
   1:  PR[GP1:91,2] = PR[GP1:90,2] + 9.095;
   1:L PR[91] 10mm/sec CNT100;
   1:  PR[GP1:91,1] = PR[GP1:90,1] + 15.061;
   1:  PR[GP1:91,2] = PR[GP1:90,2] + 9.772;
   1:L PR[91] 10mm/sec CNT100;
   1:  PR[GP1:91,1] = PR[GP1:90,1] + 13.819;
   1:  PR[GP1:91,2] = PR[GP1:90,2] + 10.132;
   1:L PR[91] 10mm/sec CNT100;
   1:  PR[GP1:91,1] = PR[GP1:90,1] + 10.281;
   1:  PR[GP1:91,2] = PR[GP1:90,2] + 10.478;
   1:L PR[91] 10mm/sec CNT100;
   1:  PR[GP1:91,1] = PR[GP1:90,1] + 9.968;
   1:  PR[GP1:91,2] = PR[GP1:90,2] + 10.452;
   1:L PR[91] 10mm/sec CNT100;
   1:  PR[GP1:91,1] = PR[GP1:90,1] + 6.696;
   1:  PR[GP1:91,2] = PR[GP1:90,2] + 10.082;
   1:L PR[91] 10mm/sec CNT100;
   1:  PR[GP1:91,1] = PR[GP1:90,1] + 6.411;
   1:  PR[GP1:91,2] = PR[GP1:90,2] + 10.034;
   1:L PR[91] 10mm/sec CNT100;
   1:  PR[GP1:91,1] = PR[GP1:90,1] + 5.570;
   1:  PR[GP1:91,2] = PR[GP1:90,2] + 9.994;
   1:L PR[91] 10mm/sec CNT100;
   1:  PR[GP1:91,1] = PR[GP1:90,1] + 4.835;
   1:  PR[GP1:91,2] = PR[GP1:90,2] + 10.035;
   1:L PR[91] 10mm/sec CNT100;
   1:  PR[GP1:91,1] = PR[GP1:90,1] + 1.906;
   1:  PR[GP1:91,2] = PR[GP1:90,2] + 10.042;
   1:L PR[91] 10mm/sec CNT100;
   1:  PR[GP1:91,1] = PR[GP1:90,1] + 0.159;
   1:  PR[GP1:91,2] = PR[GP1:90,2] + 10.091;
   1:L PR[91] 10mm/sec CNT100;
   1:  PR[GP1:91,1] = PR[GP1:90,1] + -1.698;
   1:  PR[GP1:91,2] = PR[GP1:90,2] + 9.766;
   1:L PR[91] 10mm/sec CNT100;
   1:  PR[GP1:91,1] = PR[GP1:90,1] + -4.188;
   1:  PR[GP1:91,2] = PR[GP1:90,2] + 9.403;
   1:L PR[91] 10mm/sec CNT100;
   1:  PR[GP1:91,1] = PR[GP1:90,1] + -5.143;
   1:  PR[GP1:91,2] = PR[GP1:90,2] + 9.038;
   1:L PR[91] 10mm/sec CNT100;
   1:  PR[GP1:91,1] = PR[GP1:90,1] + -8.092;
   1:  PR[GP1:91,2] = PR[GP1:90,2] + 8.013;
   1:L PR[91] 10mm/sec CNT100;
   1:  PR[GP1:91,1] = PR[GP1:90,1] + -8.356;
   1:  PR[GP1:91,2] = PR[GP1:90,2] + 7.840;
   1:L PR[91] 10mm/sec CNT100;
   1:  PR[GP1:91,1] = PR[GP1:90,1] + -10.519;
   1:  PR[GP1:91,2] = PR[GP1:90,2] + 6.523;
   1:L PR[91] 10mm/sec CNT100;
   1:  PR[GP1:91,1] = PR[GP1:90,1] + -11.445;
   1:  PR[GP1:91,2] = PR[GP1:90,2] + 5.937;
   1:L PR[91] 10mm/sec CNT100;
   1:  PR[GP1:91,1] = PR[GP1:90,1] + -13.999;
   1:  PR[GP1:91,2] = PR[GP1:90,2] + 3.327;
   1:L PR[91] 10mm/sec CNT100;
   1:  PR[GP1:91,1] = PR[GP1:90,1] + -14.178;
   1:  PR[GP1:91,2] = PR[GP1:90,2] + 3.073;
   1:L PR[91] 10mm/sec CNT100;
   1:  PR[GP1:91,1] = PR[GP1:90,1] + -15.698;
   1:  PR[GP1:91,2] = PR[GP1:90,2] + 0.414;
   1:L PR[91] 10mm/sec CNT100;
   1:  PR[GP1:91,1] = PR[GP1:90,1] + -15.879;
   1:  PR[GP1:91,2] = PR[GP1:90,2] + 0.037;
   1:L PR[91] 10mm/sec CNT100;
   1:  PR[GP1:91,1] = PR[GP1:90,1] + -16.780;
   1:  PR[GP1:91,2] = PR[GP1:90,2] + -3.188;
   1:L PR[91] 10mm/sec CNT100;
   1:  PR[GP1:91,1] = PR[GP1:90,1] + -16.811;
   1:  PR[GP1:91,2] = PR[GP1:90,2] + -3.476;
   1:L PR[91] 10mm/sec CNT100;
   1:  PR[GP1:91,1] = PR[GP1:90,1] + -16.783;
   1:  PR[GP1:91,2] = PR[GP1:90,2] + -3.788;
   1:L PR[91] 10mm/sec CNT100;
   1:  PR[GP1:91,1] = PR[GP1:90,1] + -16.686;
   1:  PR[GP1:91,2] = PR[GP1:90,2] + -6.903;
   1:L PR[91] 10mm/sec CNT100;
   1:  PR[GP1:91,1] = PR[GP1:90,1] + -16.483;
   1:  PR[GP1:91,2] = PR[GP1:90,2] + -7.823;
   1:L PR[91] 10mm/sec CNT100;
   1:  PR[GP1:91,1] = PR[GP1:90,1] + -15.455;
   1:  PR[GP1:91,2] = PR[GP1:90,2] + -11.119;
   1:L PR[91] 10mm/sec CNT100;
   1:  PR[GP1:91,1] = PR[GP1:90,1] + -15.289;
   1:  PR[GP1:91,2] = PR[GP1:90,2] + -11.515;
   1:L PR[91] 10mm/sec CNT100;
   1:  PR[GP1:91,1] = PR[GP1:90,1] + -13.246;
   1:  PR[GP1:91,2] = PR[GP1:90,2] + -14.903;
   1:L PR[91] 10mm/sec CNT100;
   1:  PR[GP1:91,1] = PR[GP1:90,1] + -12.013;
   1:  PR[GP1:91,2] = PR[GP1:90,2] + -15.879;
   1:  PR[GP1:91,3] = PR[GP1:90,3] + 52.800;
   1:L PR[91] 10mm/sec CNT100;
   1:  PR[GP1:91,1] = PR[GP1:90,1] + -9.444;
   1:  PR[GP1:91,2] = PR[GP1:90,2] + -18.717;
   1:L PR[91] 10mm/sec CNT100;
   1:  PR[GP1:91,1] = PR[GP1:90,1] + -8.195;
   1:  PR[GP1:91,2] = PR[GP1:90,2] + -19.965;
   1:L PR[91] 10mm/sec CNT100;
   1:  PR[GP1:91,1] = PR[GP1:90,1] + -5.988;
   1:  PR[GP1:91,2] = PR[GP1:90,2] + -21.625;
   1:L PR[91] 10mm/sec CNT100;
   1:  PR[GP1:91,1] = PR[GP1:90,1] + -3.286;
   1:  PR[GP1:91,2] = PR[GP1:90,2] + -23.445;
   1:L PR[91] 10mm/sec CNT100;
   1:  PR[GP1:91,1] = PR[GP1:90,1] + -2.035;
   1:  PR[GP1:91,2] = PR[GP1:90,2] + -24.074;
   1:L PR[91] 10mm/sec CNT100;
   1:  PR[GP1:91,1] = PR[GP1:90,1] + 2.518;
   1:  PR[GP1:91,2] = PR[GP1:90,2] + -26.065;
   1:L PR[91] 10mm/sec CNT100;
   1:  PR[GP1:91,1] = PR[GP1:90,1] + 7.623;
   1:  PR[GP1:91,2] = PR[GP1:90,2] + -27.559;
   1:L PR[91] 10mm/sec CNT100;
   1:  PR[GP1:91,1] = PR[GP1:90,1] + 9.586;
   1:  PR[GP1:91,2] = PR[GP1:90,2] + -27.856;
   1:L PR[91] 10mm/sec CNT100;
   1:  PR[GP1:91,1] = PR[GP1:90,1] + 12.583;
   1:  PR[GP1:91,2] = PR[GP1:90,2] + -28.145;
   1:L PR[91] 10mm/sec CNT100;
   1:  PR[GP1:91,1] = PR[GP1:90,1] + 12.883;
   1:  PR[GP1:91,2] = PR[GP1:90,2] + -28.106;
   1:L PR[91] 10mm/sec CNT100;
   1:  PR[GP1:91,1] = PR[GP1:90,1] + 13.367;
   1:  PR[GP1:91,2] = PR[GP1:90,2] + -28.089;
   1:L PR[91] 10mm/sec CNT100;
   1:  PR[GP1:91,1] = PR[GP1:90,1] + 15.335;
   1:  PR[GP1:91,2] = PR[GP1:90,2] + -28.100;
   1:L PR[91] 10mm/sec CNT100;
   1:  PR[GP1:91,1] = PR[GP1:90,1] + 17.685;
   1:  PR[GP1:91,2] = PR[GP1:90,2] + -27.941;
   1:L PR[91] 10mm/sec CNT100;
   1:  PR[GP1:91,1] = PR[GP1:90,1] + 20.420;
   1:  PR[GP1:91,2] = PR[GP1:90,2] + -27.380;
   1:L PR[91] 10mm/sec CNT100;
   1:  PR[GP1:91,1] = PR[GP1:90,1] + 22.373;
   1:  PR[GP1:91,2] = PR[GP1:90,2] + -26.667;
   1:L PR[91] 10mm/sec CNT100;
   1:  PR[GP1:91,1] = PR[GP1:90,1] + 23.033;
   1:  PR[GP1:91,2] = PR[GP1:90,2] + -26.410;
   1:L PR[91] 10mm/sec CNT100;
   1:  PR[GP1:91,1] = PR[GP1:90,1] + 24.331;
   1:  PR[GP1:91,2] = PR[GP1:90,2] + -25.649;
   1:L PR[91] 10mm/sec CNT100;
   1:  PR[GP1:91,1] = PR[GP1:90,1] + 25.544;
   1:  PR[GP1:91,2] = PR[GP1:90,2] + -24.963;
   1:L PR[91] 10mm/sec CNT100;
   1:  PR[GP1:91,1] = PR[GP1:90,1] + 26.022;
   1:  PR[GP1:91,2] = PR[GP1:90,2] + -24.576;
   1:L PR[91] 10mm/sec CNT100;
   1:  PR[GP1:91,1] = PR[GP1:90,1] + 27.503;
   1:  PR[GP1:91,2] = PR[GP1:90,2] + -23.317;
   1:L PR[91] 10mm/sec CNT100;
   1:  PR[GP1:91,1] = PR[GP1:90,1] + 28.212;
   1:  PR[GP1:91,2] = PR[GP1:90,2] + -22.538;
   1:L PR[91] 10mm/sec CNT100;
   1:  PR[GP1:91,1] = PR[GP1:90,1] + 28.976;
   1:  PR[GP1:91,2] = PR[GP1:90,2] + -21.547;
   1:L PR[91] 10mm/sec CNT100;
   1:  PR[GP1:91,1] = PR[GP1:90,1] + 29.559;
   1:  PR[GP1:91,2] = PR[GP1:90,2] + -20.694;
   1:L PR[91] 10mm/sec CNT100;
   1:  PR[GP1:91,1] = PR[GP1:90,1] + 30.140;
   1:  PR[GP1:91,2] = PR[GP1:90,2] + -19.491;
   1:L PR[91] 10mm/sec CNT100;
   1:  PR[GP1:91,1] = PR[GP1:90,1] + 30.550;
   1:  PR[GP1:91,2] = PR[GP1:90,2] + -18.695;
   1:L PR[91] 10mm/sec CNT100;
   1:  PR[GP1:91,1] = PR[GP1:90,1] + 30.802;
   1:  PR[GP1:91,2] = PR[GP1:90,2] + -18.058;
   1:L PR[91] 10mm/sec CNT100;
   1:  PR[GP1:91,1] = PR[GP1:90,1] + 31.496;
   1:  PR[GP1:91,2] = PR[GP1:90,2] + -15.399;
   1:L PR[91] 10mm/sec CNT100;
   1:  PR[GP1:91,1] = PR[GP1:90,1] + 31.761;
   1:  PR[GP1:91,2] = PR[GP1:90,2] + -12.461;
   1:L PR[91] 10mm/sec CNT100;
   1:  PR[GP1:91,1] = PR[GP1:90,1] + 31.474;
   1:  PR[GP1:91,2] = PR[GP1:90,2] + -9.538;
   1:L PR[91] 10mm/sec CNT100;
   1:  PR[GP1:91,1] = PR[GP1:90,1] + 31.041;
   1:  PR[GP1:91,2] = PR[GP1:90,2] + -7.892;
   1:L PR[91] 10mm/sec CNT100;
   1:  PR[GP1:91,1] = PR[GP1:90,1] + 30.508;
   1:  PR[GP1:91,2] = PR[GP1:90,2] + -5.676;
   1:L PR[91] 10mm/sec CNT100;
   1:  PR[GP1:91,1] = PR[GP1:90,1] + 29.971;
   1:  PR[GP1:91,2] = PR[GP1:90,2] + -4.470;
   1:L PR[91] 10mm/sec CNT100;
   1:  PR[GP1:91,1] = PR[GP1:90,1] + 28.930;
   1:  PR[GP1:91,2] = PR[GP1:90,2] + -1.946;
   1:L PR[91] 10mm/sec CNT100;
   1:  PR[GP1:91,1] = PR[GP1:90,1] + 27.445;
   1:  PR[GP1:91,2] = PR[GP1:90,2] + 0.331;
   1:L PR[91] 10mm/sec CNT100;
   1:  PR[GP1:91,1] = PR[GP1:90,1] + 26.709;
   1:  PR[GP1:91,2] = PR[GP1:90,2] + 1.524;
   1:L PR[91] 10mm/sec CNT100;
   1:  PR[GP1:91,1] = PR[GP1:90,1] + 25.301;
   1:  PR[GP1:91,2] = PR[GP1:90,2] + 3.109;
   1:L PR[91] 10mm/sec CNT100;
   1:  PR[GP1:91,1] = PR[GP1:90,1] + 23.998;
   1:  PR[GP1:91,2] = PR[GP1:90,2] + 4.544;
   1:L PR[91] 10mm/sec CNT100;
   1:  PR[GP1:91,1] = PR[GP1:90,1] + 20.886;
   1:  PR[GP1:91,2] = PR[GP1:90,2] + 6.978;
   1:L PR[91] 10mm/sec CNT100;
   1:  PR[GP1:91,1] = PR[GP1:90,1] + 17.569;
   1:  PR[GP1:91,2] = PR[GP1:90,2] + 8.736;
   1:L PR[91] 10mm/sec CNT100;
   1:  PR[GP1:91,1] = PR[GP1:90,1] + 14.060;
   1:  PR[GP1:91,2] = PR[GP1:90,2] + 9.806;
   1:L PR[91] 10mm/sec CNT100;
   1:  PR[GP1:91,1] = PR[GP1:90,1] + 10.579;
   1:  PR[GP1:91,2] = PR[GP1:90,2] + 10.150;
   1:L PR[91] 10mm/sec CNT100;
   1:  PR[GP1:91,1] = PR[GP1:90,1] + 8.984;
   1:  PR[GP1:91,2] = PR[GP1:90,2] + 10.020;
   1:L PR[91] 10mm/sec CNT100;
   1:  PR[GP1:91,1] = PR[GP1:90,1] + 6.806;
   1:  PR[GP1:91,2] = PR[GP1:90,2] + 9.778;
   1:L PR[91] 10mm/sec CNT100;
   1:  PR[GP1:91,1] = PR[GP1:90,1] + 6.048;
   1:  PR[GP1:91,2] = PR[GP1:90,2] + 9.740;
   1:L PR[91] 10mm/sec CNT100;
   1:  PR[GP1:91,1] = PR[GP1:90,1] + 5.691;
   1:  PR[GP1:91,2] = PR[GP1:90,2] + 9.755;
   1:L PR[91] 10mm/sec CNT100;
   1:  PR[GP1:91,1] = PR[GP1:90,1] + 2.303;
   1:  PR[GP1:91,2] = PR[GP1:90,2] + 9.762;
   1:L PR[91] 10mm/sec CNT100;
   1:  PR[GP1:91,1] = PR[GP1:90,1] + 0.999;
   1:  PR[GP1:91,2] = PR[GP1:90,2] + 9.799;
   1:L PR[91] 10mm/sec CNT100;
   1:  PR[GP1:91,1] = PR[GP1:90,1] + -1.296;
   1:  PR[GP1:91,2] = PR[GP1:90,2] + 9.398;
   1:L PR[91] 10mm/sec CNT100;
   1:  PR[GP1:91,1] = PR[GP1:90,1] + -3.355;
   1:  PR[GP1:91,2] = PR[GP1:90,2] + 9.098;
   1:L PR[91] 10mm/sec CNT100;
   1:  PR[GP1:91,1] = PR[GP1:90,1] + -4.718;
   1:  PR[GP1:91,2] = PR[GP1:90,2] + 8.576;
   1:L PR[91] 10mm/sec CNT100;
   1:  PR[GP1:91,1] = PR[GP1:90,1] + -7.263;
   1:  PR[GP1:91,2] = PR[GP1:90,2] + 7.692;
   1:L PR[91] 10mm/sec CNT100;
   1:  PR[GP1:91,1] = PR[GP1:90,1] + -7.889;
   1:  PR[GP1:91,2] = PR[GP1:90,2] + 7.281;
   1:L PR[91] 10mm/sec CNT100;
   1:  PR[GP1:91,1] = PR[GP1:90,1] + -10.584;
   1:  PR[GP1:91,2] = PR[GP1:90,2] + 5.640;
   1:L PR[91] 10mm/sec CNT100;
   1:  PR[GP1:91,1] = PR[GP1:90,1] + -13.190;
   1:  PR[GP1:91,2] = PR[GP1:90,2] + 2.976;
   1:L PR[91] 10mm/sec CNT100;
   1:  PR[GP1:91,1] = PR[GP1:90,1] + -14.930;
   1:  PR[GP1:91,2] = PR[GP1:90,2] + -0.068;
   1:L PR[91] 10mm/sec CNT100;
   1:  PR[GP1:91,1] = PR[GP1:90,1] + -14.968;
   1:  PR[GP1:91,2] = PR[GP1:90,2] + -0.147;
   1:L PR[91] 10mm/sec CNT100;
   1:  PR[GP1:91,1] = PR[GP1:90,1] + -15.913;
   1:  PR[GP1:91,2] = PR[GP1:90,2] + -3.546;
   1:L PR[91] 10mm/sec CNT100;
   1:  PR[GP1:91,1] = PR[GP1:90,1] + -15.915;
   1:  PR[GP1:91,2] = PR[GP1:90,2] + -3.572;
   1:L PR[91] 10mm/sec CNT100;
   1:  PR[GP1:91,1] = PR[GP1:90,1] + -15.796;
   1:  PR[GP1:91,2] = PR[GP1:90,2] + -7.235;
   1:L PR[91] 10mm/sec CNT100;
   1:  PR[GP1:91,1] = PR[GP1:90,1] + -15.676;
   1:  PR[GP1:91,2] = PR[GP1:90,2] + -7.818;
   1:L PR[91] 10mm/sec CNT100;
   1:  PR[GP1:91,1] = PR[GP1:90,1] + -14.504;
   1:  PR[GP1:91,2] = PR[GP1:90,2] + -11.577;
   1:L PR[91] 10mm/sec CNT100;
   1:  PR[GP1:91,1] = PR[GP1:90,1] + -14.471;
   1:  PR[GP1:91,2] = PR[GP1:90,2] + -11.656;
   1:L PR[91] 10mm/sec CNT100;
   1:  PR[GP1:91,1] = PR[GP1:90,1] + -13.821;
   1:  PR[GP1:91,2] = PR[GP1:90,2] + -12.735;
   1:L PR[91] 10mm/sec CNT100;
   1:  PR[GP1:91,1] = PR[GP1:90,1] + -12.305;
   1:  PR[GP1:91,2] = PR[GP1:90,2] + -15.422;
   1:L PR[91] 10mm/sec CNT100;
   1:  PR[GP1:91,1] = PR[GP1:90,1] + -11.063;
   1:  PR[GP1:91,2] = PR[GP1:90,2] + -16.354;
   1:  PR[GP1:91,3] = PR[GP1:90,3] + 53.900;
   1:L PR[91] 10mm/sec CNT100;
   1:  PR[GP1:91,1] = PR[GP1:90,1] + -8.837;
   1:  PR[GP1:91,2] = PR[GP1:90,2] + -18.814;
   1:L PR[91] 10mm/sec CNT100;
   1:  PR[GP1:91,1] = PR[GP1:90,1] + -7.202;
   1:  PR[GP1:91,2] = PR[GP1:90,2] + -20.448;
   1:L PR[91] 10mm/sec CNT100;
   1:  PR[GP1:91,1] = PR[GP1:90,1] + -5.426;
   1:  PR[GP1:91,2] = PR[GP1:90,2] + -21.783;
   1:L PR[91] 10mm/sec CNT100;
   1:  PR[GP1:91,1] = PR[GP1:90,1] + -2.247;
   1:  PR[GP1:91,2] = PR[GP1:90,2] + -23.926;
   1:L PR[91] 10mm/sec CNT100;
   1:  PR[GP1:91,1] = PR[GP1:90,1] + -1.499;
   1:  PR[GP1:91,2] = PR[GP1:90,2] + -24.301;
   1:L PR[91] 10mm/sec CNT100;
   1:  PR[GP1:91,1] = PR[GP1:90,1] + 1.108;
   1:  PR[GP1:91,2] = PR[GP1:90,2] + -25.438;
   1:L PR[91] 10mm/sec CNT100;
   1:  PR[GP1:91,1] = PR[GP1:90,1] + 3.192;
   1:  PR[GP1:91,2] = PR[GP1:90,2] + -26.476;
   1:L PR[91] 10mm/sec CNT100;
   1:  PR[GP1:91,1] = PR[GP1:90,1] + 3.980;
   1:  PR[GP1:91,2] = PR[GP1:90,2] + -26.742;
   1:L PR[91] 10mm/sec CNT100;
   1:  PR[GP1:91,1] = PR[GP1:90,1] + 8.353;
   1:  PR[GP1:91,2] = PR[GP1:90,2] + -28.022;
   1:L PR[91] 10mm/sec CNT100;
   1:  PR[GP1:91,1] = PR[GP1:90,1] + 11.039;
   1:  PR[GP1:91,2] = PR[GP1:90,2] + -28.429;
   1:L PR[91] 10mm/sec CNT100;
   1:  PR[GP1:91,1] = PR[GP1:90,1] + 13.330;
   1:  PR[GP1:91,2] = PR[GP1:90,2] + -28.650;
   1:L PR[91] 10mm/sec CNT100;
   1:  PR[GP1:91,1] = PR[GP1:90,1] + 13.551;
   1:  PR[GP1:91,2] = PR[GP1:90,2] + -28.621;
   1:L PR[91] 10mm/sec CNT100;
   1:  PR[GP1:91,1] = PR[GP1:90,1] + 13.935;
   1:  PR[GP1:91,2] = PR[GP1:90,2] + -28.607;
   1:L PR[91] 10mm/sec CNT100;
   1:  PR[GP1:91,1] = PR[GP1:90,1] + 15.166;
   1:  PR[GP1:91,2] = PR[GP1:90,2] + -28.611;
   1:L PR[91] 10mm/sec CNT100;
   1:  PR[GP1:91,1] = PR[GP1:90,1] + 17.161;
   1:  PR[GP1:91,2] = PR[GP1:90,2] + -28.536;
   1:L PR[91] 10mm/sec CNT100;
   1:  PR[GP1:91,1] = PR[GP1:90,1] + 17.987;
   1:  PR[GP1:91,2] = PR[GP1:90,2] + -28.491;
   1:L PR[91] 10mm/sec CNT100;
   1:  PR[GP1:91,1] = PR[GP1:90,1] + 20.792;
   1:  PR[GP1:91,2] = PR[GP1:90,2] + -27.972;
   1:L PR[91] 10mm/sec CNT100;
   1:  PR[GP1:91,1] = PR[GP1:90,1] + 22.516;
   1:  PR[GP1:91,2] = PR[GP1:90,2] + -27.372;
   1:L PR[91] 10mm/sec CNT100;
   1:  PR[GP1:91,1] = PR[GP1:90,1] + 23.131;
   1:  PR[GP1:91,2] = PR[GP1:90,2] + -27.191;
   1:L PR[91] 10mm/sec CNT100;
   1:  PR[GP1:91,1] = PR[GP1:90,1] + 24.204;
   1:  PR[GP1:91,2] = PR[GP1:90,2] + -26.720;
   1:L PR[91] 10mm/sec CNT100;
   1:  PR[GP1:91,1] = PR[GP1:90,1] + 24.711;
   1:  PR[GP1:91,2] = PR[GP1:90,2] + -26.439;
   1:L PR[91] 10mm/sec CNT100;
   1:  PR[GP1:91,1] = PR[GP1:90,1] + 26.263;
   1:  PR[GP1:91,2] = PR[GP1:90,2] + -25.526;
   1:L PR[91] 10mm/sec CNT100;
   1:  PR[GP1:91,1] = PR[GP1:90,1] + 28.055;
   1:  PR[GP1:91,2] = PR[GP1:90,2] + -24.151;
   1:L PR[91] 10mm/sec CNT100;
   1:  PR[GP1:91,1] = PR[GP1:90,1] + 29.504;
   1:  PR[GP1:91,2] = PR[GP1:90,2] + -22.621;
   1:L PR[91] 10mm/sec CNT100;
   1:  PR[GP1:91,1] = PR[GP1:90,1] + 30.476;
   1:  PR[GP1:91,2] = PR[GP1:90,2] + -21.225;
   1:L PR[91] 10mm/sec CNT100;
   1:  PR[GP1:91,1] = PR[GP1:90,1] + 30.560;
   1:  PR[GP1:91,2] = PR[GP1:90,2] + -21.084;
   1:L PR[91] 10mm/sec CNT100;
   1:  PR[GP1:91,1] = PR[GP1:90,1] + 31.244;
   1:  PR[GP1:91,2] = PR[GP1:90,2] + -19.745;
   1:L PR[91] 10mm/sec CNT100;
   1:  PR[GP1:91,1] = PR[GP1:90,1] + 31.760;
   1:  PR[GP1:91,2] = PR[GP1:90,2] + -18.328;
   1:L PR[91] 10mm/sec CNT100;
   1:  PR[GP1:91,1] = PR[GP1:90,1] + 32.066;
   1:  PR[GP1:91,2] = PR[GP1:90,2] + -17.114;
   1:L PR[91] 10mm/sec CNT100;
   1:  PR[GP1:91,1] = PR[GP1:90,1] + 32.271;
   1:  PR[GP1:91,2] = PR[GP1:90,2] + -15.926;
   1:L PR[91] 10mm/sec CNT100;
   1:  PR[GP1:91,1] = PR[GP1:90,1] + 32.421;
   1:  PR[GP1:91,2] = PR[GP1:90,2] + -14.547;
   1:L PR[91] 10mm/sec CNT100;
   1:  PR[GP1:91,1] = PR[GP1:90,1] + 32.494;
   1:  PR[GP1:91,2] = PR[GP1:90,2] + -13.323;
   1:L PR[91] 10mm/sec CNT100;
   1:  PR[GP1:91,1] = PR[GP1:90,1] + 32.488;
   1:  PR[GP1:91,2] = PR[GP1:90,2] + -12.722;
   1:L PR[91] 10mm/sec CNT100;
   1:  PR[GP1:91,1] = PR[GP1:90,1] + 32.306;
   1:  PR[GP1:91,2] = PR[GP1:90,2] + -11.454;
   1:L PR[91] 10mm/sec CNT100;
   1:  PR[GP1:91,1] = PR[GP1:90,1] + 32.142;
   1:  PR[GP1:91,2] = PR[GP1:90,2] + -9.876;
   1:L PR[91] 10mm/sec CNT100;
   1:  PR[GP1:91,1] = PR[GP1:90,1] + 31.705;
   1:  PR[GP1:91,2] = PR[GP1:90,2] + -8.381;
   1:L PR[91] 10mm/sec CNT100;
   1:  PR[GP1:91,1] = PR[GP1:90,1] + 31.088;
   1:  PR[GP1:91,2] = PR[GP1:90,2] + -6.058;
   1:L PR[91] 10mm/sec CNT100;
   1:  PR[GP1:91,1] = PR[GP1:90,1] + 29.455;
   1:  PR[GP1:91,2] = PR[GP1:90,2] + -2.381;
   1:L PR[91] 10mm/sec CNT100;
   1:  PR[GP1:91,1] = PR[GP1:90,1] + 27.201;
   1:  PR[GP1:91,2] = PR[GP1:90,2] + 1.077;
   1:L PR[91] 10mm/sec CNT100;
   1:  PR[GP1:91,1] = PR[GP1:90,1] + 26.190;
   1:  PR[GP1:91,2] = PR[GP1:90,2] + 2.161;
   1:L PR[91] 10mm/sec CNT100;
   1:  PR[GP1:91,1] = PR[GP1:90,1] + 24.439;
   1:  PR[GP1:91,2] = PR[GP1:90,2] + 4.118;
   1:L PR[91] 10mm/sec CNT100;
   1:  PR[GP1:91,1] = PR[GP1:90,1] + 22.973;
   1:  PR[GP1:91,2] = PR[GP1:90,2] + 5.279;
   1:L PR[91] 10mm/sec CNT100;
   1:  PR[GP1:91,1] = PR[GP1:90,1] + 21.307;
   1:  PR[GP1:91,2] = PR[GP1:90,2] + 6.572;
   1:L PR[91] 10mm/sec CNT100;
   1:  PR[GP1:91,1] = PR[GP1:90,1] + 17.901;
   1:  PR[GP1:91,2] = PR[GP1:90,2] + 8.369;
   1:L PR[91] 10mm/sec CNT100;
   1:  PR[GP1:91,1] = PR[GP1:90,1] + 14.390;
   1:  PR[GP1:91,2] = PR[GP1:90,2] + 9.456;
   1:L PR[91] 10mm/sec CNT100;
   1:  PR[GP1:91,1] = PR[GP1:90,1] + 13.445;
   1:  PR[GP1:91,2] = PR[GP1:90,2] + 9.568;
   1:L PR[91] 10mm/sec CNT100;
   1:  PR[GP1:91,1] = PR[GP1:90,1] + 10.873;
   1:  PR[GP1:91,2] = PR[GP1:90,2] + 9.822;
   1:L PR[91] 10mm/sec CNT100;
   1:  PR[GP1:91,1] = PR[GP1:90,1] + 9.291;
   1:  PR[GP1:91,2] = PR[GP1:90,2] + 9.710;
   1:L PR[91] 10mm/sec CNT100;
   1:  PR[GP1:91,1] = PR[GP1:90,1] + 7.242;
   1:  PR[GP1:91,2] = PR[GP1:90,2] + 9.507;
   1:L PR[91] 10mm/sec CNT100;
   1:  PR[GP1:91,1] = PR[GP1:90,1] + 6.550;
   1:  PR[GP1:91,2] = PR[GP1:90,2] + 9.475;
   1:L PR[91] 10mm/sec CNT100;
   1:  PR[GP1:91,1] = PR[GP1:90,1] + 2.701;
   1:  PR[GP1:91,2] = PR[GP1:90,2] + 9.483;
   1:L PR[91] 10mm/sec CNT100;
   1:  PR[GP1:91,1] = PR[GP1:90,1] + 1.840;
   1:  PR[GP1:91,2] = PR[GP1:90,2] + 9.507;
   1:L PR[91] 10mm/sec CNT100;
   1:  PR[GP1:91,1] = PR[GP1:90,1] + -0.894;
   1:  PR[GP1:91,2] = PR[GP1:90,2] + 9.030;
   1:L PR[91] 10mm/sec CNT100;
   1:  PR[GP1:91,1] = PR[GP1:90,1] + -2.522;
   1:  PR[GP1:91,2] = PR[GP1:90,2] + 8.792;
   1:L PR[91] 10mm/sec CNT100;
   1:  PR[GP1:91,1] = PR[GP1:90,1] + -4.293;
   1:  PR[GP1:91,2] = PR[GP1:90,2] + 8.114;
   1:L PR[91] 10mm/sec CNT100;
   1:  PR[GP1:91,1] = PR[GP1:90,1] + -6.433;
   1:  PR[GP1:91,2] = PR[GP1:90,2] + 7.371;
   1:L PR[91] 10mm/sec CNT100;
   1:  PR[GP1:91,1] = PR[GP1:90,1] + -7.422;
   1:  PR[GP1:91,2] = PR[GP1:90,2] + 6.721;
   1:L PR[91] 10mm/sec CNT100;
   1:  PR[GP1:91,1] = PR[GP1:90,1] + -9.744;
   1:  PR[GP1:91,2] = PR[GP1:90,2] + 5.307;
   1:L PR[91] 10mm/sec CNT100;
   1:  PR[GP1:91,1] = PR[GP1:90,1] + -10.183;
   1:  PR[GP1:91,2] = PR[GP1:90,2] + 4.830;
   1:L PR[91] 10mm/sec CNT100;
   1:  PR[GP1:91,1] = PR[GP1:90,1] + -12.319;
   1:  PR[GP1:91,2] = PR[GP1:90,2] + 2.673;
   1:L PR[91] 10mm/sec CNT100;
   1:  PR[GP1:91,1] = PR[GP1:90,1] + -12.461;
   1:  PR[GP1:91,2] = PR[GP1:90,2] + 2.403;
   1:L PR[91] 10mm/sec CNT100;
   1:  PR[GP1:91,1] = PR[GP1:90,1] + -14.095;
   1:  PR[GP1:91,2] = PR[GP1:90,2] + -0.445;
   1:L PR[91] 10mm/sec CNT100;
   1:  PR[GP1:91,1] = PR[GP1:90,1] + -15.036;
   1:  PR[GP1:91,2] = PR[GP1:90,2] + -3.879;
   1:L PR[91] 10mm/sec CNT100;
   1:  PR[GP1:91,1] = PR[GP1:90,1] + -14.947;
   1:  PR[GP1:91,2] = PR[GP1:90,2] + -7.147;
   1:L PR[91] 10mm/sec CNT100;
   1:  PR[GP1:91,1] = PR[GP1:90,1] + -14.914;
   1:  PR[GP1:91,2] = PR[GP1:90,2] + -7.595;
   1:L PR[91] 10mm/sec CNT100;
   1:  PR[GP1:91,1] = PR[GP1:90,1] + -14.871;
   1:  PR[GP1:91,2] = PR[GP1:90,2] + -7.808;
   1:L PR[91] 10mm/sec CNT100;
   1:  PR[GP1:91,1] = PR[GP1:90,1] + -14.136;
   1:  PR[GP1:91,2] = PR[GP1:90,2] + -10.163;
   1:L PR[91] 10mm/sec CNT100;
   1:  PR[GP1:91,1] = PR[GP1:90,1] + -13.810;
   1:  PR[GP1:91,2] = PR[GP1:90,2] + -11.258;
   1:L PR[91] 10mm/sec CNT100;
   1:  PR[GP1:91,1] = PR[GP1:90,1] + -13.586;
   1:  PR[GP1:91,2] = PR[GP1:90,2] + -12.001;
   1:L PR[91] 10mm/sec CNT100;
   1:  PR[GP1:91,1] = PR[GP1:90,1] + -11.629;
   1:  PR[GP1:91,2] = PR[GP1:90,2] + -15.469;
   1:L PR[91] 10mm/sec CNT100;
   1:  PR[GP1:91,1] = PR[GP1:90,1] + -10.114;
   1:  PR[GP1:91,2] = PR[GP1:90,2] + -16.829;
   1:  PR[GP1:91,3] = PR[GP1:90,3] + 55.000;
   1:L PR[91] 10mm/sec CNT100;
   1:  PR[GP1:91,1] = PR[GP1:90,1] + -8.230;
   1:  PR[GP1:91,2] = PR[GP1:90,2] + -18.911;
   1:L PR[91] 10mm/sec CNT100;
   1:  PR[GP1:91,1] = PR[GP1:90,1] + -6.209;
   1:  PR[GP1:91,2] = PR[GP1:90,2] + -20.930;
   1:L PR[91] 10mm/sec CNT100;
   1:  PR[GP1:91,1] = PR[GP1:90,1] + -4.864;
   1:  PR[GP1:91,2] = PR[GP1:90,2] + -21.942;
   1:L PR[91] 10mm/sec CNT100;
   1:  PR[GP1:91,1] = PR[GP1:90,1] + -1.207;
   1:  PR[GP1:91,2] = PR[GP1:90,2] + -24.406;
   1:L PR[91] 10mm/sec CNT100;
   1:  PR[GP1:91,1] = PR[GP1:90,1] + -0.963;
   1:  PR[GP1:91,2] = PR[GP1:90,2] + -24.528;
   1:L PR[91] 10mm/sec CNT100;
   1:  PR[GP1:91,1] = PR[GP1:90,1] + 0.005;
   1:  PR[GP1:91,2] = PR[GP1:90,2] + -24.951;
   1:L PR[91] 10mm/sec CNT100;
   1:  PR[GP1:91,1] = PR[GP1:90,1] + 3.940;
   1:  PR[GP1:91,2] = PR[GP1:90,2] + -26.912;
   1:L PR[91] 10mm/sec CNT100;
   1:  PR[GP1:91,1] = PR[GP1:90,1] + 5.469;
   1:  PR[GP1:91,2] = PR[GP1:90,2] + -27.428;
   1:L PR[91] 10mm/sec CNT100;
   1:  PR[GP1:91,1] = PR[GP1:90,1] + 9.082;
   1:  PR[GP1:91,2] = PR[GP1:90,2] + -28.485;
   1:L PR[91] 10mm/sec CNT100;
   1:  PR[GP1:91,1] = PR[GP1:90,1] + 12.493;
   1:  PR[GP1:91,2] = PR[GP1:90,2] + -29.002;
   1:L PR[91] 10mm/sec CNT100;
   1:  PR[GP1:91,1] = PR[GP1:90,1] + 14.102;
   1:  PR[GP1:91,2] = PR[GP1:90,2] + -29.157;
   1:L PR[91] 10mm/sec CNT100;
   1:  PR[GP1:91,1] = PR[GP1:90,1] + 14.186;
   1:  PR[GP1:91,2] = PR[GP1:90,2] + -29.137;
   1:L PR[91] 10mm/sec CNT100;
   1:  PR[GP1:91,1] = PR[GP1:90,1] + 14.502;
   1:  PR[GP1:91,2] = PR[GP1:90,2] + -29.126;
   1:L PR[91] 10mm/sec CNT100;
   1:  PR[GP1:91,1] = PR[GP1:90,1] + 16.621;
   1:  PR[GP1:91,2] = PR[GP1:90,2] + -29.124;
   1:L PR[91] 10mm/sec CNT100;
   1:  PR[GP1:91,1] = PR[GP1:90,1] + 18.276;
   1:  PR[GP1:91,2] = PR[GP1:90,2] + -29.043;
   1:L PR[91] 10mm/sec CNT100;
   1:  PR[GP1:91,1] = PR[GP1:90,1] + 18.779;
   1:  PR[GP1:91,2] = PR[GP1:90,2] + -28.951;
   1:L PR[91] 10mm/sec CNT100;
   1:  PR[GP1:91,1] = PR[GP1:90,1] + 19.313;
   1:  PR[GP1:91,2] = PR[GP1:90,2] + -28.895;
   1:L PR[91] 10mm/sec CNT100;
   1:  PR[GP1:91,1] = PR[GP1:90,1] + 20.296;
   1:  PR[GP1:91,2] = PR[GP1:90,2] + -28.762;
   1:L PR[91] 10mm/sec CNT100;
   1:  PR[GP1:91,1] = PR[GP1:90,1] + 21.628;
   1:  PR[GP1:91,2] = PR[GP1:90,2] + -28.477;
   1:L PR[91] 10mm/sec CNT100;
   1:  PR[GP1:91,1] = PR[GP1:90,1] + 23.419;
   1:  PR[GP1:91,2] = PR[GP1:90,2] + -27.967;
   1:L PR[91] 10mm/sec CNT100;
   1:  PR[GP1:91,1] = PR[GP1:90,1] + 25.428;
   1:  PR[GP1:91,2] = PR[GP1:90,2] + -27.156;
   1:L PR[91] 10mm/sec CNT100;
   1:  PR[GP1:91,1] = PR[GP1:90,1] + 27.152;
   1:  PR[GP1:91,2] = PR[GP1:90,2] + -26.202;
   1:L PR[91] 10mm/sec CNT100;
   1:  PR[GP1:91,1] = PR[GP1:90,1] + 27.502;
   1:  PR[GP1:91,2] = PR[GP1:90,2] + -25.964;
   1:L PR[91] 10mm/sec CNT100;
   1:  PR[GP1:91,1] = PR[GP1:90,1] + 29.028;
   1:  PR[GP1:91,2] = PR[GP1:90,2] + -24.793;
   1:L PR[91] 10mm/sec CNT100;
   1:  PR[GP1:91,1] = PR[GP1:90,1] + 30.575;
   1:  PR[GP1:91,2] = PR[GP1:90,2] + -23.164;
   1:L PR[91] 10mm/sec CNT100;
   1:  PR[GP1:91,1] = PR[GP1:90,1] + 31.384;
   1:  PR[GP1:91,2] = PR[GP1:90,2] + -22.002;
   1:L PR[91] 10mm/sec CNT100;
   1:  PR[GP1:91,1] = PR[GP1:90,1] + 31.706;
   1:  PR[GP1:91,2] = PR[GP1:90,2] + -21.469;
   1:L PR[91] 10mm/sec CNT100;
   1:  PR[GP1:91,1] = PR[GP1:90,1] + 32.274;
   1:  PR[GP1:91,2] = PR[GP1:90,2] + -20.356;
   1:L PR[91] 10mm/sec CNT100;
   1:  PR[GP1:91,1] = PR[GP1:90,1] + 32.675;
   1:  PR[GP1:91,2] = PR[GP1:90,2] + -19.263;
   1:L PR[91] 10mm/sec CNT100;
   1:  PR[GP1:91,1] = PR[GP1:90,1] + 32.855;
   1:  PR[GP1:91,2] = PR[GP1:90,2] + -18.724;
   1:L PR[91] 10mm/sec CNT100;
   1:  PR[GP1:91,1] = PR[GP1:90,1] + 33.111;
   1:  PR[GP1:91,2] = PR[GP1:90,2] + -17.704;
   1:L PR[91] 10mm/sec CNT100;
   1:  PR[GP1:91,1] = PR[GP1:90,1] + 33.270;
   1:  PR[GP1:91,2] = PR[GP1:90,2] + -16.688;
   1:L PR[91] 10mm/sec CNT100;
   1:  PR[GP1:91,1] = PR[GP1:90,1] + 33.310;
   1:  PR[GP1:91,2] = PR[GP1:90,2] + -16.316;
   1:L PR[91] 10mm/sec CNT100;
   1:  PR[GP1:91,1] = PR[GP1:90,1] + 33.385;
   1:  PR[GP1:91,2] = PR[GP1:90,2] + -14.459;
   1:L PR[91] 10mm/sec CNT100;
   1:  PR[GP1:91,1] = PR[GP1:90,1] + 33.254;
   1:  PR[GP1:91,2] = PR[GP1:90,2] + -12.696;
   1:L PR[91] 10mm/sec CNT100;
   1:  PR[GP1:91,1] = PR[GP1:90,1] + 33.006;
   1:  PR[GP1:91,2] = PR[GP1:90,2] + -10.904;
   1:L PR[91] 10mm/sec CNT100;
   1:  PR[GP1:91,1] = PR[GP1:90,1] + 32.825;
   1:  PR[GP1:91,2] = PR[GP1:90,2] + -10.071;
   1:L PR[91] 10mm/sec CNT100;
   1:  PR[GP1:91,1] = PR[GP1:90,1] + 32.674;
   1:  PR[GP1:91,2] = PR[GP1:90,2] + -9.607;
   1:L PR[91] 10mm/sec CNT100;
   1:  PR[GP1:91,1] = PR[GP1:90,1] + 32.633;
   1:  PR[GP1:91,2] = PR[GP1:90,2] + -9.536;
   1:L PR[91] 10mm/sec CNT100;
   1:  PR[GP1:91,1] = PR[GP1:90,1] + 32.266;
   1:  PR[GP1:91,2] = PR[GP1:90,2] + -8.334;
   1:L PR[91] 10mm/sec CNT100;
   1:  PR[GP1:91,1] = PR[GP1:90,1] + 31.965;
   1:  PR[GP1:91,2] = PR[GP1:90,2] + -7.328;
   1:L PR[91] 10mm/sec CNT100;
   1:  PR[GP1:91,1] = PR[GP1:90,1] + 31.714;
   1:  PR[GP1:91,2] = PR[GP1:90,2] + -6.396;
   1:L PR[91] 10mm/sec CNT100;
   1:  PR[GP1:91,1] = PR[GP1:90,1] + 30.767;
   1:  PR[GP1:91,2] = PR[GP1:90,2] + -4.432;
   1:L PR[91] 10mm/sec CNT100;
   1:  PR[GP1:91,1] = PR[GP1:90,1] + 30.020;
   1:  PR[GP1:91,2] = PR[GP1:90,2] + -2.756;
   1:L PR[91] 10mm/sec CNT100;
   1:  PR[GP1:91,1] = PR[GP1:90,1] + 28.643;
   1:  PR[GP1:91,2] = PR[GP1:90,2] + -0.761;
   1:L PR[91] 10mm/sec CNT100;
   1:  PR[GP1:91,1] = PR[GP1:90,1] + 27.716;
   1:  PR[GP1:91,2] = PR[GP1:90,2] + 0.662;
   1:L PR[91] 10mm/sec CNT100;
   1:  PR[GP1:91,1] = PR[GP1:90,1] + 24.897;
   1:  PR[GP1:91,2] = PR[GP1:90,2] + 3.686;
   1:L PR[91] 10mm/sec CNT100;
   1:  PR[GP1:91,1] = PR[GP1:90,1] + 21.736;
   1:  PR[GP1:91,2] = PR[GP1:90,2] + 6.167;
   1:L PR[91] 10mm/sec CNT100;
   1:  PR[GP1:91,1] = PR[GP1:90,1] + 18.309;
   1:  PR[GP1:91,2] = PR[GP1:90,2] + 7.985;
   1:L PR[91] 10mm/sec CNT100;
   1:  PR[GP1:91,1] = PR[GP1:90,1] + 14.751;
   1:  PR[GP1:91,2] = PR[GP1:90,2] + 9.098;
   1:L PR[91] 10mm/sec CNT100;
   1:  PR[GP1:91,1] = PR[GP1:90,1] + 12.524;
   1:  PR[GP1:91,2] = PR[GP1:90,2] + 9.361;
   1:L PR[91] 10mm/sec CNT100;
   1:  PR[GP1:91,1] = PR[GP1:90,1] + 11.171;
   1:  PR[GP1:91,2] = PR[GP1:90,2] + 9.495;
   1:L PR[91] 10mm/sec CNT100;
   1:  PR[GP1:91,1] = PR[GP1:90,1] + 8.870;
   1:  PR[GP1:91,2] = PR[GP1:90,2] + 9.332;
   1:L PR[91] 10mm/sec CNT100;
   1:  PR[GP1:91,1] = PR[GP1:90,1] + 7.710;
   1:  PR[GP1:91,2] = PR[GP1:90,2] + 9.221;
   1:L PR[91] 10mm/sec CNT100;
   1:  PR[GP1:91,1] = PR[GP1:90,1] + 7.069;
   1:  PR[GP1:91,2] = PR[GP1:90,2] + 9.194;
   1:L PR[91] 10mm/sec CNT100;
   1:  PR[GP1:91,1] = PR[GP1:90,1] + 3.098;
   1:  PR[GP1:91,2] = PR[GP1:90,2] + 9.204;
   1:L PR[91] 10mm/sec CNT100;
   1:  PR[GP1:91,1] = PR[GP1:90,1] + 2.680;
   1:  PR[GP1:91,2] = PR[GP1:90,2] + 9.216;
   1:L PR[91] 10mm/sec CNT100;
   1:  PR[GP1:91,1] = PR[GP1:90,1] + -0.491;
   1:  PR[GP1:91,2] = PR[GP1:90,2] + 8.662;
   1:L PR[91] 10mm/sec CNT100;
   1:  PR[GP1:91,1] = PR[GP1:90,1] + -1.689;
   1:  PR[GP1:91,2] = PR[GP1:90,2] + 8.487;
   1:L PR[91] 10mm/sec CNT100;
   1:  PR[GP1:91,1] = PR[GP1:90,1] + -3.868;
   1:  PR[GP1:91,2] = PR[GP1:90,2] + 7.653;
   1:L PR[91] 10mm/sec CNT100;
   1:  PR[GP1:91,1] = PR[GP1:90,1] + -5.603;
   1:  PR[GP1:91,2] = PR[GP1:90,2] + 7.050;
   1:L PR[91] 10mm/sec CNT100;
   1:  PR[GP1:91,1] = PR[GP1:90,1] + -6.955;
   1:  PR[GP1:91,2] = PR[GP1:90,2] + 6.161;
   1:L PR[91] 10mm/sec CNT100;
   1:  PR[GP1:91,1] = PR[GP1:90,1] + -8.914;
   1:  PR[GP1:91,2] = PR[GP1:90,2] + 4.969;
   1:L PR[91] 10mm/sec CNT100;
   1:  PR[GP1:91,1] = PR[GP1:90,1] + -9.651;
   1:  PR[GP1:91,2] = PR[GP1:90,2] + 4.169;
   1:L PR[91] 10mm/sec CNT100;
   1:  PR[GP1:91,1] = PR[GP1:90,1] + -11.483;
   1:  PR[GP1:91,2] = PR[GP1:90,2] + 2.318;
   1:L PR[91] 10mm/sec CNT100;
   1:  PR[GP1:91,1] = PR[GP1:90,1] + -11.839;
   1:  PR[GP1:91,2] = PR[GP1:90,2] + 1.639;
   1:L PR[91] 10mm/sec CNT100;
   1:  PR[GP1:91,1] = PR[GP1:90,1] + -13.242;
   1:  PR[GP1:91,2] = PR[GP1:90,2] + -0.807;
   1:L PR[91] 10mm/sec CNT100;
   1:  PR[GP1:91,1] = PR[GP1:90,1] + -13.391;
   1:  PR[GP1:91,2] = PR[GP1:90,2] + -1.450;
   1:L PR[91] 10mm/sec CNT100;
   1:  PR[GP1:91,1] = PR[GP1:90,1] + -14.172;
   1:  PR[GP1:91,2] = PR[GP1:90,2] + -4.271;
   1:L PR[91] 10mm/sec CNT100;
   1:  PR[GP1:91,1] = PR[GP1:90,1] + -14.097;
   1:  PR[GP1:91,2] = PR[GP1:90,2] + -7.067;
   1:L PR[91] 10mm/sec CNT100;
   1:  PR[GP1:91,1] = PR[GP1:90,1] + -14.032;
   1:  PR[GP1:91,2] = PR[GP1:90,2] + -7.946;
   1:L PR[91] 10mm/sec CNT100;
   1:  PR[GP1:91,1] = PR[GP1:90,1] + -13.374;
   1:  PR[GP1:91,2] = PR[GP1:90,2] + -10.156;
   1:L PR[91] 10mm/sec CNT100;
   1:  PR[GP1:91,1] = PR[GP1:90,1] + -12.897;
   1:  PR[GP1:91,2] = PR[GP1:90,2] + -11.834;
   1:L PR[91] 10mm/sec CNT100;
   1:  PR[GP1:91,1] = PR[GP1:90,1] + -12.686;
   1:  PR[GP1:91,2] = PR[GP1:90,2] + -12.446;
   1:L PR[91] 10mm/sec CNT100;
   1:  PR[GP1:91,1] = PR[GP1:90,1] + -10.954;
   1:  PR[GP1:91,2] = PR[GP1:90,2] + -15.517;
   1:L PR[91] 10mm/sec CNT100;
   1:  PR[GP1:91,1] = PR[GP1:90,1] + -9.165;
   1:  PR[GP1:91,2] = PR[GP1:90,2] + -17.304;
   1:  PR[GP1:91,3] = PR[GP1:90,3] + 56.100;
   1:L PR[91] 10mm/sec CNT100;
   1:  PR[GP1:91,1] = PR[GP1:90,1] + -7.623;
   1:  PR[GP1:91,2] = PR[GP1:90,2] + -19.008;
   1:L PR[91] 10mm/sec CNT100;
   1:  PR[GP1:91,1] = PR[GP1:90,1] + -5.215;
   1:  PR[GP1:91,2] = PR[GP1:90,2] + -21.413;
   1:L PR[91] 10mm/sec CNT100;
   1:  PR[GP1:91,1] = PR[GP1:90,1] + -4.302;
   1:  PR[GP1:91,2] = PR[GP1:90,2] + -22.100;
   1:L PR[91] 10mm/sec CNT100;
   1:  PR[GP1:91,1] = PR[GP1:90,1] + -0.931;
   1:  PR[GP1:91,2] = PR[GP1:90,2] + -24.372;
   1:L PR[91] 10mm/sec CNT100;
   1:  PR[GP1:91,1] = PR[GP1:90,1] + -0.256;
   1:  PR[GP1:91,2] = PR[GP1:90,2] + -24.874;
   1:L PR[91] 10mm/sec CNT100;
   1:  PR[GP1:91,1] = PR[GP1:90,1] + -0.017;
   1:  PR[GP1:91,2] = PR[GP1:90,2] + -25.002;
   1:L PR[91] 10mm/sec CNT100;
   1:  PR[GP1:91,1] = PR[GP1:90,1] + 4.689;
   1:  PR[GP1:91,2] = PR[GP1:90,2] + -27.347;
   1:L PR[91] 10mm/sec CNT100;
   1:  PR[GP1:91,1] = PR[GP1:90,1] + 6.958;
   1:  PR[GP1:91,2] = PR[GP1:90,2] + -28.113;
   1:L PR[91] 10mm/sec CNT100;
   1:  PR[GP1:91,1] = PR[GP1:90,1] + 9.812;
   1:  PR[GP1:91,2] = PR[GP1:90,2] + -28.948;
   1:L PR[91] 10mm/sec CNT100;
   1:  PR[GP1:91,1] = PR[GP1:90,1] + 13.946;
   1:  PR[GP1:91,2] = PR[GP1:90,2] + -29.575;
   1:L PR[91] 10mm/sec CNT100;
   1:  PR[GP1:91,1] = PR[GP1:90,1] + 14.868;
   1:  PR[GP1:91,2] = PR[GP1:90,2] + -29.664;
   1:L PR[91] 10mm/sec CNT100;
   1:  PR[GP1:91,1] = PR[GP1:90,1] + 15.047;
   1:  PR[GP1:91,2] = PR[GP1:90,2] + -29.645;
   1:L PR[91] 10mm/sec CNT100;
   1:  PR[GP1:91,1] = PR[GP1:90,1] + 16.295;
   1:  PR[GP1:91,2] = PR[GP1:90,2] + -29.644;
   1:L PR[91] 10mm/sec CNT100;
   1:  PR[GP1:91,1] = PR[GP1:90,1] + 17.868;
   1:  PR[GP1:91,2] = PR[GP1:90,2] + -29.563;
   1:L PR[91] 10mm/sec CNT100;
   1:  PR[GP1:91,1] = PR[GP1:90,1] + 18.070;
   1:  PR[GP1:91,2] = PR[GP1:90,2] + -29.540;
   1:L PR[91] 10mm/sec CNT100;
   1:  PR[GP1:91,1] = PR[GP1:90,1] + 19.770;
   1:  PR[GP1:91,2] = PR[GP1:90,2] + -29.558;
   1:L PR[91] 10mm/sec CNT100;
   1:  PR[GP1:91,1] = PR[GP1:90,1] + 20.030;
   1:  PR[GP1:91,2] = PR[GP1:90,2] + -29.536;
   1:L PR[91] 10mm/sec CNT100;
   1:  PR[GP1:91,1] = PR[GP1:90,1] + 21.167;
   1:  PR[GP1:91,2] = PR[GP1:90,2] + -29.374;
   1:L PR[91] 10mm/sec CNT100;
   1:  PR[GP1:91,1] = PR[GP1:90,1] + 22.440;
   1:  PR[GP1:91,2] = PR[GP1:90,2] + -29.117;
   1:L PR[91] 10mm/sec CNT100;
   1:  PR[GP1:91,1] = PR[GP1:90,1] + 22.879;
   1:  PR[GP1:91,2] = PR[GP1:90,2] + -29.012;
   1:L PR[91] 10mm/sec CNT100;
   1:  PR[GP1:91,1] = PR[GP1:90,1] + 24.405;
   1:  PR[GP1:91,2] = PR[GP1:90,2] + -28.577;
   1:L PR[91] 10mm/sec CNT100;
   1:  PR[GP1:91,1] = PR[GP1:90,1] + 25.001;
   1:  PR[GP1:91,2] = PR[GP1:90,2] + -28.322;
   1:L PR[91] 10mm/sec CNT100;
   1:  PR[GP1:91,1] = PR[GP1:90,1] + 26.585;
   1:  PR[GP1:91,2] = PR[GP1:90,2] + -27.685;
   1:L PR[91] 10mm/sec CNT100;
   1:  PR[GP1:91,1] = PR[GP1:90,1] + 28.019;
   1:  PR[GP1:91,2] = PR[GP1:90,2] + -26.892;
   1:L PR[91] 10mm/sec CNT100;
   1:  PR[GP1:91,1] = PR[GP1:90,1] + 28.761;
   1:  PR[GP1:91,2] = PR[GP1:90,2] + -26.387;
   1:L PR[91] 10mm/sec CNT100;
   1:  PR[GP1:91,1] = PR[GP1:90,1] + 30.002;
   1:  PR[GP1:91,2] = PR[GP1:90,2] + -25.435;
   1:L PR[91] 10mm/sec CNT100;
   1:  PR[GP1:91,1] = PR[GP1:90,1] + 31.646;
   1:  PR[GP1:91,2] = PR[GP1:90,2] + -23.707;
   1:L PR[91] 10mm/sec CNT100;
   1:  PR[GP1:91,1] = PR[GP1:90,1] + 32.291;
   1:  PR[GP1:91,2] = PR[GP1:90,2] + -22.780;
   1:L PR[91] 10mm/sec CNT100;
   1:  PR[GP1:91,1] = PR[GP1:90,1] + 32.851;
   1:  PR[GP1:91,2] = PR[GP1:90,2] + -21.855;
   1:L PR[91] 10mm/sec CNT100;
   1:  PR[GP1:91,1] = PR[GP1:90,1] + 33.304;
   1:  PR[GP1:91,2] = PR[GP1:90,2] + -20.967;
   1:L PR[91] 10mm/sec CNT100;
   1:  PR[GP1:91,1] = PR[GP1:90,1] + 33.624;
   1:  PR[GP1:91,2] = PR[GP1:90,2] + -20.095;
   1:L PR[91] 10mm/sec CNT100;
   1:  PR[GP1:91,1] = PR[GP1:90,1] + 33.951;
   1:  PR[GP1:91,2] = PR[GP1:90,2] + -19.111;
   1:L PR[91] 10mm/sec CNT100;
   1:  PR[GP1:91,1] = PR[GP1:90,1] + 34.158;
   1:  PR[GP1:91,2] = PR[GP1:90,2] + -18.289;
   1:L PR[91] 10mm/sec CNT100;
   1:  PR[GP1:91,1] = PR[GP1:90,1] + 34.286;
   1:  PR[GP1:91,2] = PR[GP1:90,2] + -17.469;
   1:L PR[91] 10mm/sec CNT100;
   1:  PR[GP1:91,1] = PR[GP1:90,1] + 34.377;
   1:  PR[GP1:91,2] = PR[GP1:90,2] + -16.618;
   1:L PR[91] 10mm/sec CNT100;
   1:  PR[GP1:91,1] = PR[GP1:90,1] + 34.440;
   1:  PR[GP1:91,2] = PR[GP1:90,2] + -15.085;
   1:L PR[91] 10mm/sec CNT100;
   1:  PR[GP1:91,1] = PR[GP1:90,1] + 34.275;
   1:  PR[GP1:91,2] = PR[GP1:90,2] + -13.115;
   1:L PR[91] 10mm/sec CNT100;
   1:  PR[GP1:91,1] = PR[GP1:90,1] + 34.047;
   1:  PR[GP1:91,2] = PR[GP1:90,2] + -11.852;
   1:L PR[91] 10mm/sec CNT100;
   1:  PR[GP1:91,1] = PR[GP1:90,1] + 33.744;
   1:  PR[GP1:91,2] = PR[GP1:90,2] + -10.682;
   1:L PR[91] 10mm/sec CNT100;
   1:  PR[GP1:91,1] = PR[GP1:90,1] + 33.603;
   1:  PR[GP1:91,2] = PR[GP1:90,2] + -10.209;
   1:L PR[91] 10mm/sec CNT100;
   1:  PR[GP1:91,1] = PR[GP1:90,1] + 33.210;
   1:  PR[GP1:91,2] = PR[GP1:90,2] + -9.187;
   1:L PR[91] 10mm/sec CNT100;
   1:  PR[GP1:91,1] = PR[GP1:90,1] + 32.950;
   1:  PR[GP1:91,2] = PR[GP1:90,2] + -8.398;
   1:L PR[91] 10mm/sec CNT100;
   1:  PR[GP1:91,1] = PR[GP1:90,1] + 32.828;
   1:  PR[GP1:91,2] = PR[GP1:90,2] + -8.189;
   1:L PR[91] 10mm/sec CNT100;
   1:  PR[GP1:91,1] = PR[GP1:90,1] + 32.389;
   1:  PR[GP1:91,2] = PR[GP1:90,2] + -6.752;
   1:L PR[91] 10mm/sec CNT100;
   1:  PR[GP1:91,1] = PR[GP1:90,1] + 31.894;
   1:  PR[GP1:91,2] = PR[GP1:90,2] + -5.805;
   1:L PR[91] 10mm/sec CNT100;
   1:  PR[GP1:91,1] = PR[GP1:90,1] + 30.604;
   1:  PR[GP1:91,2] = PR[GP1:90,2] + -3.125;
   1:L PR[91] 10mm/sec CNT100;
   1:  PR[GP1:91,1] = PR[GP1:90,1] + 30.285;
   1:  PR[GP1:91,2] = PR[GP1:90,2] + -2.690;
   1:L PR[91] 10mm/sec CNT100;
   1:  PR[GP1:91,1] = PR[GP1:90,1] + 29.238;
   1:  PR[GP1:91,2] = PR[GP1:90,2] + -1.191;
   1:L PR[91] 10mm/sec CNT100;
   1:  PR[GP1:91,1] = PR[GP1:90,1] + 28.250;
   1:  PR[GP1:91,2] = PR[GP1:90,2] + 0.255;
   1:L PR[91] 10mm/sec CNT100;
   1:  PR[GP1:91,1] = PR[GP1:90,1] + 27.634;
   1:  PR[GP1:91,2] = PR[GP1:90,2] + 0.887;
   1:L PR[91] 10mm/sec CNT100;
   1:  PR[GP1:91,1] = PR[GP1:90,1] + 25.403;
   1:  PR[GP1:91,2] = PR[GP1:90,2] + 3.279;
   1:L PR[91] 10mm/sec CNT100;
   1:  PR[GP1:91,1] = PR[GP1:90,1] + 22.171;
   1:  PR[GP1:91,2] = PR[GP1:90,2] + 5.758;
   1:L PR[91] 10mm/sec CNT100;
   1:  PR[GP1:91,1] = PR[GP1:90,1] + 18.716;
   1:  PR[GP1:91,2] = PR[GP1:90,2] + 7.601;
   1:L PR[91] 10mm/sec CNT100;
   1:  PR[GP1:91,1] = PR[GP1:90,1] + 15.113;
   1:  PR[GP1:91,2] = PR[GP1:90,2] + 8.739;
   1:L PR[91] 10mm/sec CNT100;
   1:  PR[GP1:91,1] = PR[GP1:90,1] + 11.464;
   1:  PR[GP1:91,2] = PR[GP1:90,2] + 9.166;
   1:L PR[91] 10mm/sec CNT100;
   1:  PR[GP1:91,1] = PR[GP1:90,1] + 8.190;
   1:  PR[GP1:91,2] = PR[GP1:90,2] + 8.929;
   1:L PR[91] 10mm/sec CNT100;
   1:  PR[GP1:91,1] = PR[GP1:90,1] + 7.610;
   1:  PR[GP1:91,2] = PR[GP1:90,2] + 8.903;
   1:L PR[91] 10mm/sec CNT100;
   1:  PR[GP1:91,1] = PR[GP1:90,1] + 3.528;
   1:  PR[GP1:91,2] = PR[GP1:90,2] + 8.925;
   1:L PR[91] 10mm/sec CNT100;
   1:  PR[GP1:91,1] = PR[GP1:90,1] + -0.089;
   1:  PR[GP1:91,2] = PR[GP1:90,2] + 8.293;
   1:L PR[91] 10mm/sec CNT100;
   1:  PR[GP1:91,1] = PR[GP1:90,1] + -0.856;
   1:  PR[GP1:91,2] = PR[GP1:90,2] + 8.182;
   1:L PR[91] 10mm/sec CNT100;
   1:  PR[GP1:91,1] = PR[GP1:90,1] + -3.444;
   1:  PR[GP1:91,2] = PR[GP1:90,2] + 7.191;
   1:L PR[91] 10mm/sec CNT100;
   1:  PR[GP1:91,1] = PR[GP1:90,1] + -4.773;
   1:  PR[GP1:91,2] = PR[GP1:90,2] + 6.729;
   1:L PR[91] 10mm/sec CNT100;
   1:  PR[GP1:91,1] = PR[GP1:90,1] + -6.488;
   1:  PR[GP1:91,2] = PR[GP1:90,2] + 5.602;
   1:L PR[91] 10mm/sec CNT100;
   1:  PR[GP1:91,1] = PR[GP1:90,1] + -8.083;
   1:  PR[GP1:91,2] = PR[GP1:90,2] + 4.631;
   1:L PR[91] 10mm/sec CNT100;
   1:  PR[GP1:91,1] = PR[GP1:90,1] + -9.118;
   1:  PR[GP1:91,2] = PR[GP1:90,2] + 3.507;
   1:L PR[91] 10mm/sec CNT100;
   1:  PR[GP1:91,1] = PR[GP1:90,1] + -10.647;
   1:  PR[GP1:91,2] = PR[GP1:90,2] + 1.962;
   1:L PR[91] 10mm/sec CNT100;
   1:  PR[GP1:91,1] = PR[GP1:90,1] + -11.217;
   1:  PR[GP1:91,2] = PR[GP1:90,2] + 0.875;
   1:L PR[91] 10mm/sec CNT100;
   1:  PR[GP1:91,1] = PR[GP1:90,1] + -12.396;
   1:  PR[GP1:91,2] = PR[GP1:90,2] + -1.180;
   1:L PR[91] 10mm/sec CNT100;
   1:  PR[GP1:91,1] = PR[GP1:90,1] + -12.658;
   1:  PR[GP1:91,2] = PR[GP1:90,2] + -2.311;
   1:L PR[91] 10mm/sec CNT100;
   1:  PR[GP1:91,1] = PR[GP1:90,1] + -13.309;
   1:  PR[GP1:91,2] = PR[GP1:90,2] + -4.662;
   1:L PR[91] 10mm/sec CNT100;
   1:  PR[GP1:91,1] = PR[GP1:90,1] + -13.246;
   1:  PR[GP1:91,2] = PR[GP1:90,2] + -6.987;
   1:L PR[91] 10mm/sec CNT100;
   1:  PR[GP1:91,1] = PR[GP1:90,1] + -13.197;
   1:  PR[GP1:91,2] = PR[GP1:90,2] + -7.654;
   1:L PR[91] 10mm/sec CNT100;
   1:  PR[GP1:91,1] = PR[GP1:90,1] + -13.150;
   1:  PR[GP1:91,2] = PR[GP1:90,2] + -8.344;
   1:L PR[91] 10mm/sec CNT100;
   1:  PR[GP1:91,1] = PR[GP1:90,1] + -12.311;
   1:  PR[GP1:91,2] = PR[GP1:90,2] + -11.219;
   1:L PR[91] 10mm/sec CNT100;
   1:  PR[GP1:91,1] = PR[GP1:90,1] + -12.145;
   1:  PR[GP1:91,2] = PR[GP1:90,2] + -11.846;
   1:L PR[91] 10mm/sec CNT100;
   1:  PR[GP1:91,1] = PR[GP1:90,1] + -11.779;
   1:  PR[GP1:91,2] = PR[GP1:90,2] + -12.904;
   1:L PR[91] 10mm/sec CNT100;
   1:  PR[GP1:91,1] = PR[GP1:90,1] + -10.278;
   1:  PR[GP1:91,2] = PR[GP1:90,2] + -15.565;
   1:L PR[91] 10mm/sec CNT100;
   1:  PR[GP1:91,1] = PR[GP1:90,1] + -8.216;
   1:  PR[GP1:91,2] = PR[GP1:90,2] + -17.779;
   1:  PR[GP1:91,3] = PR[GP1:90,3] + 57.200;
   1:L PR[91] 10mm/sec CNT100;
   1:  PR[GP1:91,1] = PR[GP1:90,1] + -7.016;
   1:  PR[GP1:91,2] = PR[GP1:90,2] + -19.105;
   1:L PR[91] 10mm/sec CNT100;
   1:  PR[GP1:91,1] = PR[GP1:90,1] + -4.222;
   1:  PR[GP1:91,2] = PR[GP1:90,2] + -21.896;
   1:L PR[91] 10mm/sec CNT100;
   1:  PR[GP1:91,1] = PR[GP1:90,1] + -3.740;
   1:  PR[GP1:91,2] = PR[GP1:90,2] + -22.259;
   1:L PR[91] 10mm/sec CNT100;
   1:  PR[GP1:91,1] = PR[GP1:90,1] + -1.877;
   1:  PR[GP1:91,2] = PR[GP1:90,2] + -23.514;
   1:L PR[91] 10mm/sec CNT100;
   1:  PR[GP1:91,1] = PR[GP1:90,1] + 0.517;
   1:  PR[GP1:91,2] = PR[GP1:90,2] + -25.292;
   1:L PR[91] 10mm/sec CNT100;
   1:  PR[GP1:91,1] = PR[GP1:90,1] + 1.465;
   1:  PR[GP1:91,2] = PR[GP1:90,2] + -25.803;
   1:L PR[91] 10mm/sec CNT100;
   1:  PR[GP1:91,1] = PR[GP1:90,1] + 5.437;
   1:  PR[GP1:91,2] = PR[GP1:90,2] + -27.782;
   1:L PR[91] 10mm/sec CNT100;
   1:  PR[GP1:91,1] = PR[GP1:90,1] + 8.447;
   1:  PR[GP1:91,2] = PR[GP1:90,2] + -28.799;
   1:L PR[91] 10mm/sec CNT100;
   1:  PR[GP1:91,1] = PR[GP1:90,1] + 10.542;
   1:  PR[GP1:91,2] = PR[GP1:90,2] + -29.412;
   1:L PR[91] 10mm/sec CNT100;
   1:  PR[GP1:91,1] = PR[GP1:90,1] + 15.399;
   1:  PR[GP1:91,2] = PR[GP1:90,2] + -30.148;
   1:L PR[91] 10mm/sec CNT100;
   1:  PR[GP1:91,1] = PR[GP1:90,1] + 15.612;
   1:  PR[GP1:91,2] = PR[GP1:90,2] + -30.168;
   1:L PR[91] 10mm/sec CNT100;
   1:  PR[GP1:91,1] = PR[GP1:90,1] + 16.466;
   1:  PR[GP1:91,2] = PR[GP1:90,2] + -30.134;
   1:L PR[91] 10mm/sec CNT100;
   1:  PR[GP1:91,1] = PR[GP1:90,1] + 20.483;
   1:  PR[GP1:91,2] = PR[GP1:90,2] + -30.178;
   1:L PR[91] 10mm/sec CNT100;
   1:  PR[GP1:91,1] = PR[GP1:90,1] + 21.170;
   1:  PR[GP1:91,2] = PR[GP1:90,2] + -30.121;
   1:L PR[91] 10mm/sec CNT100;
   1:  PR[GP1:91,1] = PR[GP1:90,1] + 22.143;
   1:  PR[GP1:91,2] = PR[GP1:90,2] + -29.982;
   1:L PR[91] 10mm/sec CNT100;
   1:  PR[GP1:91,1] = PR[GP1:90,1] + 23.234;
   1:  PR[GP1:91,2] = PR[GP1:90,2] + -29.762;
   1:L PR[91] 10mm/sec CNT100;
   1:  PR[GP1:91,1] = PR[GP1:90,1] + 24.134;
   1:  PR[GP1:91,2] = PR[GP1:90,2] + -29.546;
   1:L PR[91] 10mm/sec CNT100;
   1:  PR[GP1:91,1] = PR[GP1:90,1] + 25.398;
   1:  PR[GP1:91,2] = PR[GP1:90,2] + -29.186;
   1:L PR[91] 10mm/sec CNT100;
   1:  PR[GP1:91,1] = PR[GP1:90,1] + 26.471;
   1:  PR[GP1:91,2] = PR[GP1:90,2] + -28.726;
   1:L PR[91] 10mm/sec CNT100;
   1:  PR[GP1:91,1] = PR[GP1:90,1] + 27.742;
   1:  PR[GP1:91,2] = PR[GP1:90,2] + -28.215;
   1:L PR[91] 10mm/sec CNT100;
   1:  PR[GP1:91,1] = PR[GP1:90,1] + 28.885;
   1:  PR[GP1:91,2] = PR[GP1:90,2] + -27.583;
   1:L PR[91] 10mm/sec CNT100;
   1:  PR[GP1:91,1] = PR[GP1:90,1] + 30.020;
   1:  PR[GP1:91,2] = PR[GP1:90,2] + -26.810;
   1:L PR[91] 10mm/sec CNT100;
   1:  PR[GP1:91,1] = PR[GP1:90,1] + 30.976;
   1:  PR[GP1:91,2] = PR[GP1:90,2] + -26.077;
   1:L PR[91] 10mm/sec CNT100;
   1:  PR[GP1:91,1] = PR[GP1:90,1] + 32.718;
   1:  PR[GP1:91,2] = PR[GP1:90,2] + -24.250;
   1:L PR[91] 10mm/sec CNT100;
   1:  PR[GP1:91,1] = PR[GP1:90,1] + 33.199;
   1:  PR[GP1:91,2] = PR[GP1:90,2] + -23.558;
   1:L PR[91] 10mm/sec CNT100;
   1:  PR[GP1:91,1] = PR[GP1:90,1] + 33.996;
   1:  PR[GP1:91,2] = PR[GP1:90,2] + -22.240;
   1:L PR[91] 10mm/sec CNT100;
   1:  PR[GP1:91,1] = PR[GP1:90,1] + 34.333;
   1:  PR[GP1:91,2] = PR[GP1:90,2] + -21.578;
   1:L PR[91] 10mm/sec CNT100;
   1:  PR[GP1:91,1] = PR[GP1:90,1] + 34.573;
   1:  PR[GP1:91,2] = PR[GP1:90,2] + -20.926;
   1:L PR[91] 10mm/sec CNT100;
   1:  PR[GP1:91,1] = PR[GP1:90,1] + 35.047;
   1:  PR[GP1:91,2] = PR[GP1:90,2] + -19.499;
   1:L PR[91] 10mm/sec CNT100;
   1:  PR[GP1:91,1] = PR[GP1:90,1] + 35.204;
   1:  PR[GP1:91,2] = PR[GP1:90,2] + -18.874;
   1:L PR[91] 10mm/sec CNT100;
   1:  PR[GP1:91,1] = PR[GP1:90,1] + 35.302;
   1:  PR[GP1:91,2] = PR[GP1:90,2] + -18.249;
   1:L PR[91] 10mm/sec CNT100;
   1:  PR[GP1:91,1] = PR[GP1:90,1] + 35.445;
   1:  PR[GP1:91,2] = PR[GP1:90,2] + -16.919;
   1:L PR[91] 10mm/sec CNT100;
   1:  PR[GP1:91,1] = PR[GP1:90,1] + 35.494;
   1:  PR[GP1:91,2] = PR[GP1:90,2] + -15.708;
   1:L PR[91] 10mm/sec CNT100;
   1:  PR[GP1:91,1] = PR[GP1:90,1] + 35.306;
   1:  PR[GP1:91,2] = PR[GP1:90,2] + -13.509;
   1:L PR[91] 10mm/sec CNT100;
   1:  PR[GP1:91,1] = PR[GP1:90,1] + 35.118;
   1:  PR[GP1:91,2] = PR[GP1:90,2] + -12.473;
   1:L PR[91] 10mm/sec CNT100;
   1:  PR[GP1:91,1] = PR[GP1:90,1] + 34.869;
   1:  PR[GP1:91,2] = PR[GP1:90,2] + -11.509;
   1:L PR[91] 10mm/sec CNT100;
   1:  PR[GP1:91,1] = PR[GP1:90,1] + 34.598;
   1:  PR[GP1:91,2] = PR[GP1:90,2] + -10.569;
   1:L PR[91] 10mm/sec CNT100;
   1:  PR[GP1:91,1] = PR[GP1:90,1] + 33.682;
   1:  PR[GP1:91,2] = PR[GP1:90,2] + -8.242;
   1:L PR[91] 10mm/sec CNT100;
   1:  PR[GP1:91,1] = PR[GP1:90,1] + 33.315;
   1:  PR[GP1:91,2] = PR[GP1:90,2] + -7.509;
   1:L PR[91] 10mm/sec CNT100;
   1:  PR[GP1:91,1] = PR[GP1:90,1] + 33.313;
   1:  PR[GP1:91,2] = PR[GP1:90,2] + -7.511;
   1:L PR[91] 10mm/sec CNT100;
   1:  PR[GP1:91,1] = PR[GP1:90,1] + 31.476;
   1:  PR[GP1:91,2] = PR[GP1:90,2] + -3.995;
   1:L PR[91] 10mm/sec CNT100;
   1:  PR[GP1:91,1] = PR[GP1:90,1] + 31.211;
   1:  PR[GP1:91,2] = PR[GP1:90,2] + -3.445;
   1:L PR[91] 10mm/sec CNT100;
   1:  PR[GP1:91,1] = PR[GP1:90,1] + 30.299;
   1:  PR[GP1:91,2] = PR[GP1:90,2] + -2.227;
   1:L PR[91] 10mm/sec CNT100;
   1:  PR[GP1:91,1] = PR[GP1:90,1] + 29.423;
   1:  PR[GP1:91,2] = PR[GP1:90,2] + -1.010;
   1:L PR[91] 10mm/sec CNT100;
   1:  PR[GP1:91,1] = PR[GP1:90,1] + 28.799;
   1:  PR[GP1:91,2] = PR[GP1:90,2] + -0.106;
   1:L PR[91] 10mm/sec CNT100;
   1:  PR[GP1:91,1] = PR[GP1:90,1] + 27.687;
   1:  PR[GP1:91,2] = PR[GP1:90,2] + 1.018;
   1:L PR[91] 10mm/sec CNT100;
   1:  PR[GP1:91,1] = PR[GP1:90,1] + 25.911;
   1:  PR[GP1:91,2] = PR[GP1:90,2] + 2.872;
   1:L PR[91] 10mm/sec CNT100;
   1:  PR[GP1:91,1] = PR[GP1:90,1] + 22.656;
   1:  PR[GP1:91,2] = PR[GP1:90,2] + 5.360;
   1:L PR[91] 10mm/sec CNT100;
   1:  PR[GP1:91,1] = PR[GP1:90,1] + 19.127;
   1:  PR[GP1:91,2] = PR[GP1:90,2] + 7.216;
   1:L PR[91] 10mm/sec CNT100;
   1:  PR[GP1:91,1] = PR[GP1:90,1] + 15.476;
   1:  PR[GP1:91,2] = PR[GP1:90,2] + 8.380;
   1:L PR[91] 10mm/sec CNT100;
   1:  PR[GP1:91,1] = PR[GP1:90,1] + 11.838;
   1:  PR[GP1:91,2] = PR[GP1:90,2] + 8.814;
   1:L PR[91] 10mm/sec CNT100;
   1:  PR[GP1:91,1] = PR[GP1:90,1] + 11.184;
   1:  PR[GP1:91,2] = PR[GP1:90,2] + 8.791;
   1:L PR[91] 10mm/sec CNT100;
   1:  PR[GP1:91,1] = PR[GP1:90,1] + 8.715;
   1:  PR[GP1:91,2] = PR[GP1:90,2] + 8.622;
   1:L PR[91] 10mm/sec CNT100;
   1:  PR[GP1:91,1] = PR[GP1:90,1] + 8.181;
   1:  PR[GP1:91,2] = PR[GP1:90,2] + 8.602;
   1:L PR[91] 10mm/sec CNT100;
   1:  PR[GP1:91,1] = PR[GP1:90,1] + 5.195;
   1:  PR[GP1:91,2] = PR[GP1:90,2] + 8.608;
   1:L PR[91] 10mm/sec CNT100;
   1:  PR[GP1:91,1] = PR[GP1:90,1] + 4.266;
   1:  PR[GP1:91,2] = PR[GP1:90,2] + 8.578;
   1:L PR[91] 10mm/sec CNT100;
   1:  PR[GP1:91,1] = PR[GP1:90,1] + 2.165;
   1:  PR[GP1:91,2] = PR[GP1:90,2] + 8.249;
   1:L PR[91] 10mm/sec CNT100;
   1:  PR[GP1:91,1] = PR[GP1:90,1] + -0.016;
   1:  PR[GP1:91,2] = PR[GP1:90,2] + 7.879;
   1:L PR[91] 10mm/sec CNT100;
   1:  PR[GP1:91,1] = PR[GP1:90,1] + -3.019;
   1:  PR[GP1:91,2] = PR[GP1:90,2] + 6.729;
   1:L PR[91] 10mm/sec CNT100;
   1:  PR[GP1:91,1] = PR[GP1:90,1] + -3.943;
   1:  PR[GP1:91,2] = PR[GP1:90,2] + 6.408;
   1:L PR[91] 10mm/sec CNT100;
   1:  PR[GP1:91,1] = PR[GP1:90,1] + -6.021;
   1:  PR[GP1:91,2] = PR[GP1:90,2] + 5.042;
   1:L PR[91] 10mm/sec CNT100;
   1:  PR[GP1:91,1] = PR[GP1:90,1] + -7.252;
   1:  PR[GP1:91,2] = PR[GP1:90,2] + 4.293;
   1:L PR[91] 10mm/sec CNT100;
   1:  PR[GP1:91,1] = PR[GP1:90,1] + -8.585;
   1:  PR[GP1:91,2] = PR[GP1:90,2] + 2.845;
   1:L PR[91] 10mm/sec CNT100;
   1:  PR[GP1:91,1] = PR[GP1:90,1] + -9.811;
   1:  PR[GP1:91,2] = PR[GP1:90,2] + 1.607;
   1:L PR[91] 10mm/sec CNT100;
   1:  PR[GP1:91,1] = PR[GP1:90,1] + -10.596;
   1:  PR[GP1:91,2] = PR[GP1:90,2] + 0.111;
   1:L PR[91] 10mm/sec CNT100;
   1:  PR[GP1:91,1] = PR[GP1:90,1] + -11.550;
   1:  PR[GP1:91,2] = PR[GP1:90,2] + -1.553;
   1:L PR[91] 10mm/sec CNT100;
   1:  PR[GP1:91,1] = PR[GP1:90,1] + -11.924;
   1:  PR[GP1:91,2] = PR[GP1:90,2] + -3.172;
   1:L PR[91] 10mm/sec CNT100;
   1:  PR[GP1:91,1] = PR[GP1:90,1] + -12.445;
   1:  PR[GP1:91,2] = PR[GP1:90,2] + -5.054;
   1:L PR[91] 10mm/sec CNT100;
   1:  PR[GP1:91,1] = PR[GP1:90,1] + -12.395;
   1:  PR[GP1:91,2] = PR[GP1:90,2] + -6.908;
   1:L PR[91] 10mm/sec CNT100;
   1:  PR[GP1:91,1] = PR[GP1:90,1] + -12.356;
   1:  PR[GP1:91,2] = PR[GP1:90,2] + -7.443;
   1:L PR[91] 10mm/sec CNT100;
   1:  PR[GP1:91,1] = PR[GP1:90,1] + -12.290;
   1:  PR[GP1:91,2] = PR[GP1:90,2] + -8.407;
   1:L PR[91] 10mm/sec CNT100;
   1:  PR[GP1:91,1] = PR[GP1:90,1] + -12.269;
   1:  PR[GP1:91,2] = PR[GP1:90,2] + -8.757;
   1:L PR[91] 10mm/sec CNT100;
   1:  PR[GP1:91,1] = PR[GP1:90,1] + -11.628;
   1:  PR[GP1:91,2] = PR[GP1:90,2] + -10.971;
   1:L PR[91] 10mm/sec CNT100;
   1:  PR[GP1:91,1] = PR[GP1:90,1] + -11.394;
   1:  PR[GP1:91,2] = PR[GP1:90,2] + -11.852;
   1:L PR[91] 10mm/sec CNT100;
   1:  PR[GP1:91,1] = PR[GP1:90,1] + -10.872;
   1:  PR[GP1:91,2] = PR[GP1:90,2] + -13.361;
   1:L PR[91] 10mm/sec CNT100;
   1:  PR[GP1:91,1] = PR[GP1:90,1] + -9.602;
   1:  PR[GP1:91,2] = PR[GP1:90,2] + -15.612;
   1:L PR[91] 10mm/sec CNT100;
   1:  PR[GP1:91,1] = PR[GP1:90,1] + -7.267;
   1:  PR[GP1:91,2] = PR[GP1:90,2] + -18.254;
   1:  PR[GP1:91,3] = PR[GP1:90,3] + 58.300;
   1:L PR[91] 10mm/sec CNT100;
   1:  PR[GP1:91,1] = PR[GP1:90,1] + -6.408;
   1:  PR[GP1:91,2] = PR[GP1:90,2] + -19.202;
   1:L PR[91] 10mm/sec CNT100;
   1:  PR[GP1:91,1] = PR[GP1:90,1] + -3.238;
   1:  PR[GP1:91,2] = PR[GP1:90,2] + -22.369;
   1:L PR[91] 10mm/sec CNT100;
   1:  PR[GP1:91,1] = PR[GP1:90,1] + -2.819;
   1:  PR[GP1:91,2] = PR[GP1:90,2] + -22.659;
   1:L PR[91] 10mm/sec CNT100;
   1:  PR[GP1:91,1] = PR[GP1:90,1] + 1.290;
   1:  PR[GP1:91,2] = PR[GP1:90,2] + -25.711;
   1:L PR[91] 10mm/sec CNT100;
   1:  PR[GP1:91,1] = PR[GP1:90,1] + 2.947;
   1:  PR[GP1:91,2] = PR[GP1:90,2] + -26.604;
   1:L PR[91] 10mm/sec CNT100;
   1:  PR[GP1:91,1] = PR[GP1:90,1] + 6.186;
   1:  PR[GP1:91,2] = PR[GP1:90,2] + -28.218;
   1:L PR[91] 10mm/sec CNT100;
   1:  PR[GP1:91,1] = PR[GP1:90,1] + 9.936;
   1:  PR[GP1:91,2] = PR[GP1:90,2] + -29.484;
   1:L PR[91] 10mm/sec CNT100;
   1:  PR[GP1:91,1] = PR[GP1:90,1] + 11.272;
   1:  PR[GP1:91,2] = PR[GP1:90,2] + -29.875;
   1:L PR[91] 10mm/sec CNT100;
   1:  PR[GP1:91,1] = PR[GP1:90,1] + 15.115;
   1:  PR[GP1:91,2] = PR[GP1:90,2] + -30.457;
   1:L PR[91] 10mm/sec CNT100;
   1:  PR[GP1:91,1] = PR[GP1:90,1] + 16.492;
   1:  PR[GP1:91,2] = PR[GP1:90,2] + -30.734;
   1:L PR[91] 10mm/sec CNT100;
   1:  PR[GP1:91,1] = PR[GP1:90,1] + 16.761;
   1:  PR[GP1:91,2] = PR[GP1:90,2] + -30.750;
   1:L PR[91] 10mm/sec CNT100;
   1:  PR[GP1:91,1] = PR[GP1:90,1] + 21.195;
   1:  PR[GP1:91,2] = PR[GP1:90,2] + -30.797;
   1:L PR[91] 10mm/sec CNT100;
   1:  PR[GP1:91,1] = PR[GP1:90,1] + 22.311;
   1:  PR[GP1:91,2] = PR[GP1:90,2] + -30.705;
   1:L PR[91] 10mm/sec CNT100;
   1:  PR[GP1:91,1] = PR[GP1:90,1] + 23.120;
   1:  PR[GP1:91,2] = PR[GP1:90,2] + -30.590;
   1:L PR[91] 10mm/sec CNT100;
   1:  PR[GP1:91,1] = PR[GP1:90,1] + 24.029;
   1:  PR[GP1:91,2] = PR[GP1:90,2] + -30.406;
   1:L PR[91] 10mm/sec CNT100;
   1:  PR[GP1:91,1] = PR[GP1:90,1] + 25.388;
   1:  PR[GP1:91,2] = PR[GP1:90,2] + -30.080;
   1:L PR[91] 10mm/sec CNT100;
   1:  PR[GP1:91,1] = PR[GP1:90,1] + 26.391;
   1:  PR[GP1:91,2] = PR[GP1:90,2] + -29.794;
   1:L PR[91] 10mm/sec CNT100;
   1:  PR[GP1:91,1] = PR[GP1:90,1] + 27.942;
   1:  PR[GP1:91,2] = PR[GP1:90,2] + -29.130;
   1:L PR[91] 10mm/sec CNT100;
   1:  PR[GP1:91,1] = PR[GP1:90,1] + 28.900;
   1:  PR[GP1:91,2] = PR[GP1:90,2] + -28.745;
   1:L PR[91] 10mm/sec CNT100;
   1:  PR[GP1:91,1] = PR[GP1:90,1] + 29.752;
   1:  PR[GP1:91,2] = PR[GP1:90,2] + -28.273;
   1:L PR[91] 10mm/sec CNT100;
   1:  PR[GP1:91,1] = PR[GP1:90,1] + 31.279;
   1:  PR[GP1:91,2] = PR[GP1:90,2] + -27.233;
   1:L PR[91] 10mm/sec CNT100;
   1:  PR[GP1:91,1] = PR[GP1:90,1] + 31.949;
   1:  PR[GP1:91,2] = PR[GP1:90,2] + -26.719;
   1:L PR[91] 10mm/sec CNT100;
   1:  PR[GP1:91,1] = PR[GP1:90,1] + 33.789;
   1:  PR[GP1:91,2] = PR[GP1:90,2] + -24.794;
   1:L PR[91] 10mm/sec CNT100;
   1:  PR[GP1:91,1] = PR[GP1:90,1] + 34.107;
   1:  PR[GP1:91,2] = PR[GP1:90,2] + -24.336;
   1:L PR[91] 10mm/sec CNT100;
   1:  PR[GP1:91,1] = PR[GP1:90,1] + 35.141;
   1:  PR[GP1:91,2] = PR[GP1:90,2] + -22.625;
   1:L PR[91] 10mm/sec CNT100;
   1:  PR[GP1:91,1] = PR[GP1:90,1] + 35.363;
   1:  PR[GP1:91,2] = PR[GP1:90,2] + -22.190;
   1:L PR[91] 10mm/sec CNT100;
   1:  PR[GP1:91,1] = PR[GP1:90,1] + 35.521;
   1:  PR[GP1:91,2] = PR[GP1:90,2] + -21.758;
   1:L PR[91] 10mm/sec CNT100;
   1:  PR[GP1:91,1] = PR[GP1:90,1] + 36.144;
   1:  PR[GP1:91,2] = PR[GP1:90,2] + -19.886;
   1:L PR[91] 10mm/sec CNT100;
   1:  PR[GP1:91,1] = PR[GP1:90,1] + 36.251;
   1:  PR[GP1:91,2] = PR[GP1:90,2] + -19.459;
   1:L PR[91] 10mm/sec CNT100;
   1:  PR[GP1:91,1] = PR[GP1:90,1] + 36.318;
   1:  PR[GP1:91,2] = PR[GP1:90,2] + -19.030;
   1:L PR[91] 10mm/sec CNT100;
   1:  PR[GP1:91,1] = PR[GP1:90,1] + 36.513;
   1:  PR[GP1:91,2] = PR[GP1:90,2] + -17.220;
   1:L PR[91] 10mm/sec CNT100;
   1:  PR[GP1:91,1] = PR[GP1:90,1] + 36.549;
   1:  PR[GP1:91,2] = PR[GP1:90,2] + -16.331;
   1:L PR[91] 10mm/sec CNT100;
   1:  PR[GP1:91,1] = PR[GP1:90,1] + 36.336;
   1:  PR[GP1:91,2] = PR[GP1:90,2] + -13.903;
   1:L PR[91] 10mm/sec CNT100;
   1:  PR[GP1:91,1] = PR[GP1:90,1] + 36.190;
   1:  PR[GP1:91,2] = PR[GP1:90,2] + -13.095;
   1:L PR[91] 10mm/sec CNT100;
   1:  PR[GP1:91,1] = PR[GP1:90,1] + 35.994;
   1:  PR[GP1:91,2] = PR[GP1:90,2] + -12.338;
   1:L PR[91] 10mm/sec CNT100;
   1:  PR[GP1:91,1] = PR[GP1:90,1] + 35.593;
   1:  PR[GP1:91,2] = PR[GP1:90,2] + -10.929;
   1:L PR[91] 10mm/sec CNT100;
   1:  PR[GP1:91,1] = PR[GP1:90,1] + 34.836;
   1:  PR[GP1:91,2] = PR[GP1:90,2] + -9.002;
   1:L PR[91] 10mm/sec CNT100;
   1:  PR[GP1:91,1] = PR[GP1:90,1] + 34.593;
   1:  PR[GP1:91,2] = PR[GP1:90,2] + -8.454;
   1:L PR[91] 10mm/sec CNT100;
   1:  PR[GP1:91,1] = PR[GP1:90,1] + 33.974;
   1:  PR[GP1:91,2] = PR[GP1:90,2] + -7.240;
   1:L PR[91] 10mm/sec CNT100;
   1:  PR[GP1:91,1] = PR[GP1:90,1] + 33.073;
   1:  PR[GP1:91,2] = PR[GP1:90,2] + -5.733;
   1:L PR[91] 10mm/sec CNT100;
   1:  PR[GP1:91,1] = PR[GP1:90,1] + 32.950;
   1:  PR[GP1:91,2] = PR[GP1:90,2] + -5.824;
   1:L PR[91] 10mm/sec CNT100;
   1:  PR[GP1:91,1] = PR[GP1:90,1] + 31.901;
   1:  PR[GP1:91,2] = PR[GP1:90,2] + -3.813;
   1:L PR[91] 10mm/sec CNT100;
   1:  PR[GP1:91,1] = PR[GP1:90,1] + 30.848;
   1:  PR[GP1:91,2] = PR[GP1:90,2] + -2.469;
   1:L PR[91] 10mm/sec CNT100;
   1:  PR[GP1:91,1] = PR[GP1:90,1] + 30.141;
   1:  PR[GP1:91,2] = PR[GP1:90,2] + -1.524;
   1:L PR[91] 10mm/sec CNT100;
   1:  PR[GP1:91,1] = PR[GP1:90,1] + 29.370;
   1:  PR[GP1:91,2] = PR[GP1:90,2] + -0.453;
   1:L PR[91] 10mm/sec CNT100;
   1:  PR[GP1:91,1] = PR[GP1:90,1] + 28.447;
   1:  PR[GP1:91,2] = PR[GP1:90,2] + 0.444;
   1:L PR[91] 10mm/sec CNT100;
   1:  PR[GP1:91,1] = PR[GP1:90,1] + 26.440;
   1:  PR[GP1:91,2] = PR[GP1:90,2] + 2.496;
   1:L PR[91] 10mm/sec CNT100;
   1:  PR[GP1:91,1] = PR[GP1:90,1] + 24.696;
   1:  PR[GP1:91,2] = PR[GP1:90,2] + 3.781;
   1:L PR[91] 10mm/sec CNT100;
   1:  PR[GP1:91,1] = PR[GP1:90,1] + 23.148;
   1:  PR[GP1:91,2] = PR[GP1:90,2] + 4.964;
   1:L PR[91] 10mm/sec CNT100;
   1:  PR[GP1:91,1] = PR[GP1:90,1] + 19.598;
   1:  PR[GP1:91,2] = PR[GP1:90,2] + 6.828;
   1:L PR[91] 10mm/sec CNT100;
   1:  PR[GP1:91,1] = PR[GP1:90,1] + 15.921;
   1:  PR[GP1:91,2] = PR[GP1:90,2] + 8.003;
   1:L PR[91] 10mm/sec CNT100;
   1:  PR[GP1:91,1] = PR[GP1:90,1] + 12.241;
   1:  PR[GP1:91,2] = PR[GP1:90,2] + 8.456;
   1:L PR[91] 10mm/sec CNT100;
   1:  PR[GP1:91,1] = PR[GP1:90,1] + 10.732;
   1:  PR[GP1:91,2] = PR[GP1:90,2] + 8.402;
   1:L PR[91] 10mm/sec CNT100;
   1:  PR[GP1:91,1] = PR[GP1:90,1] + 8.785;
   1:  PR[GP1:91,2] = PR[GP1:90,2] + 8.291;
   1:L PR[91] 10mm/sec CNT100;
   1:  PR[GP1:91,1] = PR[GP1:90,1] + 6.444;
   1:  PR[GP1:91,2] = PR[GP1:90,2] + 8.281;
   1:L PR[91] 10mm/sec CNT100;
   1:  PR[GP1:91,1] = PR[GP1:90,1] + 4.991;
   1:  PR[GP1:91,2] = PR[GP1:90,2] + 8.224;
   1:L PR[91] 10mm/sec CNT100;
   1:  PR[GP1:91,1] = PR[GP1:90,1] + 0.810;
   1:  PR[GP1:91,2] = PR[GP1:90,2] + 7.568;
   1:L PR[91] 10mm/sec CNT100;
   1:  PR[GP1:91,1] = PR[GP1:90,1] + -2.594;
   1:  PR[GP1:91,2] = PR[GP1:90,2] + 6.267;
   1:L PR[91] 10mm/sec CNT100;
   1:  PR[GP1:91,1] = PR[GP1:90,1] + -3.114;
   1:  PR[GP1:91,2] = PR[GP1:90,2] + 6.087;
   1:L PR[91] 10mm/sec CNT100;
   1:  PR[GP1:91,1] = PR[GP1:90,1] + -5.553;
   1:  PR[GP1:91,2] = PR[GP1:90,2] + 4.483;
   1:L PR[91] 10mm/sec CNT100;
   1:  PR[GP1:91,1] = PR[GP1:90,1] + -6.421;
   1:  PR[GP1:91,2] = PR[GP1:90,2] + 3.955;
   1:L PR[91] 10mm/sec CNT100;
   1:  PR[GP1:91,1] = PR[GP1:90,1] + -8.052;
   1:  PR[GP1:91,2] = PR[GP1:90,2] + 2.183;
   1:L PR[91] 10mm/sec CNT100;
   1:  PR[GP1:91,1] = PR[GP1:90,1] + -8.975;
   1:  PR[GP1:91,2] = PR[GP1:90,2] + 1.251;
   1:L PR[91] 10mm/sec CNT100;
   1:  PR[GP1:91,1] = PR[GP1:90,1] + -9.974;
   1:  PR[GP1:91,2] = PR[GP1:90,2] + -0.654;
   1:L PR[91] 10mm/sec CNT100;
   1:  PR[GP1:91,1] = PR[GP1:90,1] + -10.704;
   1:  PR[GP1:91,2] = PR[GP1:90,2] + -1.926;
   1:L PR[91] 10mm/sec CNT100;
   1:  PR[GP1:91,1] = PR[GP1:90,1] + -11.191;
   1:  PR[GP1:91,2] = PR[GP1:90,2] + -4.033;
   1:L PR[91] 10mm/sec CNT100;
   1:  PR[GP1:91,1] = PR[GP1:90,1] + -11.582;
   1:  PR[GP1:91,2] = PR[GP1:90,2] + -5.445;
   1:L PR[91] 10mm/sec CNT100;
   1:  PR[GP1:91,1] = PR[GP1:90,1] + -11.545;
   1:  PR[GP1:91,2] = PR[GP1:90,2] + -6.828;
   1:L PR[91] 10mm/sec CNT100;
   1:  PR[GP1:91,1] = PR[GP1:90,1] + -11.515;
   1:  PR[GP1:91,2] = PR[GP1:90,2] + -7.232;
   1:L PR[91] 10mm/sec CNT100;
   1:  PR[GP1:91,1] = PR[GP1:90,1] + -11.465;
   1:  PR[GP1:91,2] = PR[GP1:90,2] + -7.966;
   1:L PR[91] 10mm/sec CNT100;
   1:  PR[GP1:91,1] = PR[GP1:90,1] + -11.390;
   1:  PR[GP1:91,2] = PR[GP1:90,2] + -9.182;
   1:L PR[91] 10mm/sec CNT100;
   1:  PR[GP1:91,1] = PR[GP1:90,1] + -10.945;
   1:  PR[GP1:91,2] = PR[GP1:90,2] + -10.722;
   1:L PR[91] 10mm/sec CNT100;
   1:  PR[GP1:91,1] = PR[GP1:90,1] + -10.643;
   1:  PR[GP1:91,2] = PR[GP1:90,2] + -11.858;
   1:L PR[91] 10mm/sec CNT100;
   1:  PR[GP1:91,1] = PR[GP1:90,1] + -9.965;
   1:  PR[GP1:91,2] = PR[GP1:90,2] + -13.818;
   1:L PR[91] 10mm/sec CNT100;
   1:  PR[GP1:91,1] = PR[GP1:90,1] + -8.926;
   1:  PR[GP1:91,2] = PR[GP1:90,2] + -15.660;
   1:L PR[91] 10mm/sec CNT100;
   1:  PR[GP1:91,1] = PR[GP1:90,1] + -6.317;
   1:  PR[GP1:91,2] = PR[GP1:90,2] + -18.729;
   1:  PR[GP1:91,3] = PR[GP1:90,3] + 59.400;
   1:L PR[91] 10mm/sec CNT100;
   1:  PR[GP1:91,1] = PR[GP1:90,1] + -5.801;
   1:  PR[GP1:91,2] = PR[GP1:90,2] + -19.299;
   1:L PR[91] 10mm/sec CNT100;
   1:  PR[GP1:91,1] = PR[GP1:90,1] + -3.538;
   1:  PR[GP1:91,2] = PR[GP1:90,2] + -21.561;
   1:L PR[91] 10mm/sec CNT100;
   1:  PR[GP1:91,1] = PR[GP1:90,1] + -2.370;
   1:  PR[GP1:91,2] = PR[GP1:90,2] + -22.821;
   1:L PR[91] 10mm/sec CNT100;
   1:  PR[GP1:91,1] = PR[GP1:90,1] + -1.939;
   1:  PR[GP1:91,2] = PR[GP1:90,2] + -23.157;
   1:L PR[91] 10mm/sec CNT100;
   1:  PR[GP1:91,1] = PR[GP1:90,1] + 2.062;
   1:  PR[GP1:91,2] = PR[GP1:90,2] + -26.130;
   1:L PR[91] 10mm/sec CNT100;
   1:  PR[GP1:91,1] = PR[GP1:90,1] + 4.429;
   1:  PR[GP1:91,2] = PR[GP1:90,2] + -27.404;
   1:L PR[91] 10mm/sec CNT100;
   1:  PR[GP1:91,1] = PR[GP1:90,1] + 6.934;
   1:  PR[GP1:91,2] = PR[GP1:90,2] + -28.653;
   1:L PR[91] 10mm/sec CNT100;
   1:  PR[GP1:91,1] = PR[GP1:90,1] + 11.425;
   1:  PR[GP1:91,2] = PR[GP1:90,2] + -30.169;
   1:L PR[91] 10mm/sec CNT100;
   1:  PR[GP1:91,1] = PR[GP1:90,1] + 12.002;
   1:  PR[GP1:91,2] = PR[GP1:90,2] + -30.338;
   1:L PR[91] 10mm/sec CNT100;
   1:  PR[GP1:91,1] = PR[GP1:90,1] + 13.732;
   1:  PR[GP1:91,2] = PR[GP1:90,2] + -30.600;
   1:L PR[91] 10mm/sec CNT100;
   1:  PR[GP1:91,1] = PR[GP1:90,1] + 17.363;
   1:  PR[GP1:91,2] = PR[GP1:90,2] + -31.331;
   1:L PR[91] 10mm/sec CNT100;
   1:  PR[GP1:91,1] = PR[GP1:90,1] + 18.160;
   1:  PR[GP1:91,2] = PR[GP1:90,2] + -31.377;
   1:L PR[91] 10mm/sec CNT100;
   1:  PR[GP1:91,1] = PR[GP1:90,1] + 21.907;
   1:  PR[GP1:91,2] = PR[GP1:90,2] + -31.417;
   1:L PR[91] 10mm/sec CNT100;
   1:  PR[GP1:91,1] = PR[GP1:90,1] + 23.452;
   1:  PR[GP1:91,2] = PR[GP1:90,2] + -31.289;
   1:L PR[91] 10mm/sec CNT100;
   1:  PR[GP1:91,1] = PR[GP1:90,1] + 24.097;
   1:  PR[GP1:91,2] = PR[GP1:90,2] + -31.197;
   1:L PR[91] 10mm/sec CNT100;
   1:  PR[GP1:91,1] = PR[GP1:90,1] + 24.824;
   1:  PR[GP1:91,2] = PR[GP1:90,2] + -31.050;
   1:L PR[91] 10mm/sec CNT100;
   1:  PR[GP1:91,1] = PR[GP1:90,1] + 26.643;
   1:  PR[GP1:91,2] = PR[GP1:90,2] + -30.614;
   1:L PR[91] 10mm/sec CNT100;
   1:  PR[GP1:91,1] = PR[GP1:90,1] + 27.384;
   1:  PR[GP1:91,2] = PR[GP1:90,2] + -30.403;
   1:L PR[91] 10mm/sec CNT100;
   1:  PR[GP1:91,1] = PR[GP1:90,1] + 29.413;
   1:  PR[GP1:91,2] = PR[GP1:90,2] + -29.533;
   1:L PR[91] 10mm/sec CNT100;
   1:  PR[GP1:91,1] = PR[GP1:90,1] + 30.057;
   1:  PR[GP1:91,2] = PR[GP1:90,2] + -29.275;
   1:L PR[91] 10mm/sec CNT100;
   1:  PR[GP1:91,1] = PR[GP1:90,1] + 30.618;
   1:  PR[GP1:91,2] = PR[GP1:90,2] + -28.964;
   1:L PR[91] 10mm/sec CNT100;
   1:  PR[GP1:91,1] = PR[GP1:90,1] + 32.538;
   1:  PR[GP1:91,2] = PR[GP1:90,2] + -27.656;
   1:L PR[91] 10mm/sec CNT100;
   1:  PR[GP1:91,1] = PR[GP1:90,1] + 32.923;
   1:  PR[GP1:91,2] = PR[GP1:90,2] + -27.361;
   1:L PR[91] 10mm/sec CNT100;
   1:  PR[GP1:91,1] = PR[GP1:90,1] + 34.860;
   1:  PR[GP1:91,2] = PR[GP1:90,2] + -25.337;
   1:L PR[91] 10mm/sec CNT100;
   1:  PR[GP1:91,1] = PR[GP1:90,1] + 35.015;
   1:  PR[GP1:91,2] = PR[GP1:90,2] + -25.113;
   1:L PR[91] 10mm/sec CNT100;
   1:  PR[GP1:91,1] = PR[GP1:90,1] + 36.286;
   1:  PR[GP1:91,2] = PR[GP1:90,2] + -23.010;
   1:L PR[91] 10mm/sec CNT100;
   1:  PR[GP1:91,1] = PR[GP1:90,1] + 36.388;
   1:  PR[GP1:91,2] = PR[GP1:90,2] + -22.809;
   1:L PR[91] 10mm/sec CNT100;
   1:  PR[GP1:91,1] = PR[GP1:90,1] + 37.240;
   1:  PR[GP1:91,2] = PR[GP1:90,2] + -20.272;
   1:L PR[91] 10mm/sec CNT100;
   1:  PR[GP1:91,1] = PR[GP1:90,1] + 37.298;
   1:  PR[GP1:91,2] = PR[GP1:90,2] + -20.044;
   1:L PR[91] 10mm/sec CNT100;
   1:  PR[GP1:91,1] = PR[GP1:90,1] + 37.334;
   1:  PR[GP1:91,2] = PR[GP1:90,2] + -19.810;
   1:L PR[91] 10mm/sec CNT100;
   1:  PR[GP1:91,1] = PR[GP1:90,1] + 37.580;
   1:  PR[GP1:91,2] = PR[GP1:90,2] + -17.521;
   1:L PR[91] 10mm/sec CNT100;
   1:  PR[GP1:91,1] = PR[GP1:90,1] + 37.603;
   1:  PR[GP1:91,2] = PR[GP1:90,2] + -16.954;
   1:L PR[91] 10mm/sec CNT100;
   1:  PR[GP1:91,1] = PR[GP1:90,1] + 37.367;
   1:  PR[GP1:91,2] = PR[GP1:90,2] + -14.298;
   1:L PR[91] 10mm/sec CNT100;
   1:  PR[GP1:91,1] = PR[GP1:90,1] + 37.262;
   1:  PR[GP1:91,2] = PR[GP1:90,2] + -13.716;
   1:L PR[91] 10mm/sec CNT100;
   1:  PR[GP1:91,1] = PR[GP1:90,1] + 37.119;
   1:  PR[GP1:91,2] = PR[GP1:90,2] + -13.167;
   1:L PR[91] 10mm/sec CNT100;
   1:  PR[GP1:91,1] = PR[GP1:90,1] + 36.589;
   1:  PR[GP1:91,2] = PR[GP1:90,2] + -11.289;
   1:L PR[91] 10mm/sec CNT100;
   1:  PR[GP1:91,1] = PR[GP1:90,1] + 35.996;
   1:  PR[GP1:91,2] = PR[GP1:90,2] + -9.776;
   1:L PR[91] 10mm/sec CNT100;
   1:  PR[GP1:91,1] = PR[GP1:90,1] + 35.570;
   1:  PR[GP1:91,2] = PR[GP1:90,2] + -8.817;
   1:L PR[91] 10mm/sec CNT100;
   1:  PR[GP1:91,1] = PR[GP1:90,1] + 35.060;
   1:  PR[GP1:91,2] = PR[GP1:90,2] + -7.814;
   1:L PR[91] 10mm/sec CNT100;
   1:  PR[GP1:91,1] = PR[GP1:90,1] + 33.973;
   1:  PR[GP1:91,2] = PR[GP1:90,2] + -5.997;
   1:L PR[91] 10mm/sec CNT100;
   1:  PR[GP1:91,1] = PR[GP1:90,1] + 32.825;
   1:  PR[GP1:91,2] = PR[GP1:90,2] + -4.379;
   1:L PR[91] 10mm/sec CNT100;
   1:  PR[GP1:91,1] = PR[GP1:90,1] + 32.588;
   1:  PR[GP1:91,2] = PR[GP1:90,2] + -4.085;
   1:L PR[91] 10mm/sec CNT100;
   1:  PR[GP1:91,1] = PR[GP1:90,1] + 32.553;
   1:  PR[GP1:91,2] = PR[GP1:90,2] + -4.109;
   1:L PR[91] 10mm/sec CNT100;
   1:  PR[GP1:91,1] = PR[GP1:90,1] + 31.203;
   1:  PR[GP1:91,2] = PR[GP1:90,2] + -2.402;
   1:L PR[91] 10mm/sec CNT100;
   1:  PR[GP1:91,1] = PR[GP1:90,1] + 29.957;
   1:  PR[GP1:91,2] = PR[GP1:90,2] + -0.782;
   1:L PR[91] 10mm/sec CNT100;
   1:  PR[GP1:91,1] = PR[GP1:90,1] + 28.607;
   1:  PR[GP1:91,2] = PR[GP1:90,2] + 0.504;
   1:L PR[91] 10mm/sec CNT100;
   1:  PR[GP1:91,1] = PR[GP1:90,1] + 26.972;
   1:  PR[GP1:91,2] = PR[GP1:90,2] + 2.133;
   1:L PR[91] 10mm/sec CNT100;
   1:  PR[GP1:91,1] = PR[GP1:90,1] + 25.313;
   1:  PR[GP1:91,2] = PR[GP1:90,2] + 3.337;
   1:L PR[91] 10mm/sec CNT100;
   1:  PR[GP1:91,1] = PR[GP1:90,1] + 23.649;
   1:  PR[GP1:91,2] = PR[GP1:90,2] + 4.576;
   1:L PR[91] 10mm/sec CNT100;
   1:  PR[GP1:91,1] = PR[GP1:90,1] + 20.075;
   1:  PR[GP1:91,2] = PR[GP1:90,2] + 6.439;
   1:L PR[91] 10mm/sec CNT100;
   1:  PR[GP1:91,1] = PR[GP1:90,1] + 16.365;
   1:  PR[GP1:91,2] = PR[GP1:90,2] + 7.626;
   1:L PR[91] 10mm/sec CNT100;
   1:  PR[GP1:91,1] = PR[GP1:90,1] + 12.641;
   1:  PR[GP1:91,2] = PR[GP1:90,2] + 8.098;
   1:L PR[91] 10mm/sec CNT100;
   1:  PR[GP1:91,1] = PR[GP1:90,1] + 11.140;
   1:  PR[GP1:91,2] = PR[GP1:90,2] + 8.053;
   1:L PR[91] 10mm/sec CNT100;
   1:  PR[GP1:91,1] = PR[GP1:90,1] + 9.831;
   1:  PR[GP1:91,2] = PR[GP1:90,2] + 7.986;
   1:L PR[91] 10mm/sec CNT100;
   1:  PR[GP1:91,1] = PR[GP1:90,1] + 7.950;
   1:  PR[GP1:91,2] = PR[GP1:90,2] + 7.957;
   1:L PR[91] 10mm/sec CNT100;
   1:  PR[GP1:91,1] = PR[GP1:90,1] + 5.714;
   1:  PR[GP1:91,2] = PR[GP1:90,2] + 7.870;
   1:L PR[91] 10mm/sec CNT100;
   1:  PR[GP1:91,1] = PR[GP1:90,1] + 2.124;
   1:  PR[GP1:91,2] = PR[GP1:90,2] + 7.308;
   1:L PR[91] 10mm/sec CNT100;
   1:  PR[GP1:91,1] = PR[GP1:90,1] + 1.608;
   1:  PR[GP1:91,2] = PR[GP1:90,2] + 7.204;
   1:L PR[91] 10mm/sec CNT100;
   1:  PR[GP1:91,1] = PR[GP1:90,1] + -2.278;
   1:  PR[GP1:91,2] = PR[GP1:90,2] + 5.769;
   1:L PR[91] 10mm/sec CNT100;
   1:  PR[GP1:91,1] = PR[GP1:90,1] + -5.086;
   1:  PR[GP1:91,2] = PR[GP1:90,2] + 3.923;
   1:L PR[91] 10mm/sec CNT100;
   1:  PR[GP1:91,1] = PR[GP1:90,1] + -5.590;
   1:  PR[GP1:91,2] = PR[GP1:90,2] + 3.617;
   1:L PR[91] 10mm/sec CNT100;
   1:  PR[GP1:91,1] = PR[GP1:90,1] + -7.520;
   1:  PR[GP1:91,2] = PR[GP1:90,2] + 1.521;
   1:L PR[91] 10mm/sec CNT100;
   1:  PR[GP1:91,1] = PR[GP1:90,1] + -8.139;
   1:  PR[GP1:91,2] = PR[GP1:90,2] + 0.896;
   1:L PR[91] 10mm/sec CNT100;
   1:  PR[GP1:91,1] = PR[GP1:90,1] + -9.352;
   1:  PR[GP1:91,2] = PR[GP1:90,2] + -1.418;
   1:L PR[91] 10mm/sec CNT100;
   1:  PR[GP1:91,1] = PR[GP1:90,1] + -9.858;
   1:  PR[GP1:91,2] = PR[GP1:90,2] + -2.299;
   1:L PR[91] 10mm/sec CNT100;
   1:  PR[GP1:91,1] = PR[GP1:90,1] + -10.458;
   1:  PR[GP1:91,2] = PR[GP1:90,2] + -4.894;
   1:L PR[91] 10mm/sec CNT100;
   1:  PR[GP1:91,1] = PR[GP1:90,1] + -10.719;
   1:  PR[GP1:91,2] = PR[GP1:90,2] + -5.836;
   1:L PR[91] 10mm/sec CNT100;
   1:  PR[GP1:91,1] = PR[GP1:90,1] + -10.694;
   1:  PR[GP1:91,2] = PR[GP1:90,2] + -6.748;
   1:L PR[91] 10mm/sec CNT100;
   1:  PR[GP1:91,1] = PR[GP1:90,1] + -10.674;
   1:  PR[GP1:91,2] = PR[GP1:90,2] + -7.021;
   1:L PR[91] 10mm/sec CNT100;
   1:  PR[GP1:91,1] = PR[GP1:90,1] + -10.640;
   1:  PR[GP1:91,2] = PR[GP1:90,2] + -7.526;
   1:L PR[91] 10mm/sec CNT100;
   1:  PR[GP1:91,1] = PR[GP1:90,1] + -10.512;
   1:  PR[GP1:91,2] = PR[GP1:90,2] + -9.608;
   1:L PR[91] 10mm/sec CNT100;
   1:  PR[GP1:91,1] = PR[GP1:90,1] + -10.261;
   1:  PR[GP1:91,2] = PR[GP1:90,2] + -10.473;
   1:L PR[91] 10mm/sec CNT100;
   1:  PR[GP1:91,1] = PR[GP1:90,1] + -9.893;
   1:  PR[GP1:91,2] = PR[GP1:90,2] + -11.864;
   1:L PR[91] 10mm/sec CNT100;
   1:  PR[GP1:91,1] = PR[GP1:90,1] + -9.058;
   1:  PR[GP1:91,2] = PR[GP1:90,2] + -14.276;
   1:L PR[91] 10mm/sec CNT100;
   1:  PR[GP1:91,1] = PR[GP1:90,1] + -8.250;
   1:  PR[GP1:91,2] = PR[GP1:90,2] + -15.708;
   1:L PR[91] 10mm/sec CNT100;
   1:  PR[GP1:91,1] = PR[GP1:90,1] + -5.368;
   1:  PR[GP1:91,2] = PR[GP1:90,2] + -19.204;
